// TIA Portal V18 export
FUNCTION_BLOCK "ST10_Flow6_ToolCodeScan"   // FB1076, GRAPH
// stored: AcknowledgeErrorsRequired false, AutoNumber false, GraphVersion 6.0, InitialValuesAcquisition false, SetENOAutomatically false
   // inherited from GRAPH_BASE
   VAR_INPUT
      iSysInface : "RCS_SysComInterface_V1";
   END_VAR
   VAR_IN_OUT
      ioPM_Inface : "RCS_PMInterface_V1";
      ioStatus : Int;
   END_VAR
   VAR
      sCtrlMode { S7_SetPoint := 'True'} : "SysFlowCtrlGraph";
      sUpdMES_Data : Bool;   // 更新MES数据
      工件放行中 : Bool;
      前站站号 { ExternalAccessible := 'False'; ExternalVisible := 'False'; ExternalWritable := 'False'} : UInt;
      本站站号 { ExternalAccessible := 'False'; ExternalVisible := 'False'; ExternalWritable := 'False'} : UInt;
      弹窗Temp : Array[1..10] of Int;
      AlarmID : Int;
      TON { S7_SetPoint := 'True'} : Array[0..10] of TON_TIME;
      TOF { S7_SetPoint := 'True'} : Array[0..10] of TOF_TIME;
      sUP { S7_SetPoint := 'True'} : Array[0..10] of Bool;
      更新RFID完成 : Bool;
   END_VAR
   VAR_TEMP
      Tempresult : USInt;
      本站站号乘10 : UInt;
   END_VAR
   // // TON[0] : 托盘流入1托盘到位传感器 / iA-Rotating product Check
   // // TON[1] : 托盘流入1托盘到位传感器
   // // TON[2] : 托盘流入1产品有无传感器
   // // TON[3] : 托盘流入1产品有无传感器
   // // TON[4] : 托盘流入1姿态检测光电2
   // // TON[5] : 托盘流入1姿态检测光电3
   // // TON[0].Q : 托盘流入1托盘到位 / iA-Rotating product Check
   // // TON[1].Q : 托盘流入1托盘无
   // // TON[2].Q : 托盘流入1有产品
   // // TON[3].Q : 托盘流入1无产品
   // // TON[4].Q : 托盘流入1姿态检测光电2
   // // TON[5].Q : 托盘流入1姿态检测光电3
   // // TOF[1] : iA-Rotating product Check
BEGIN
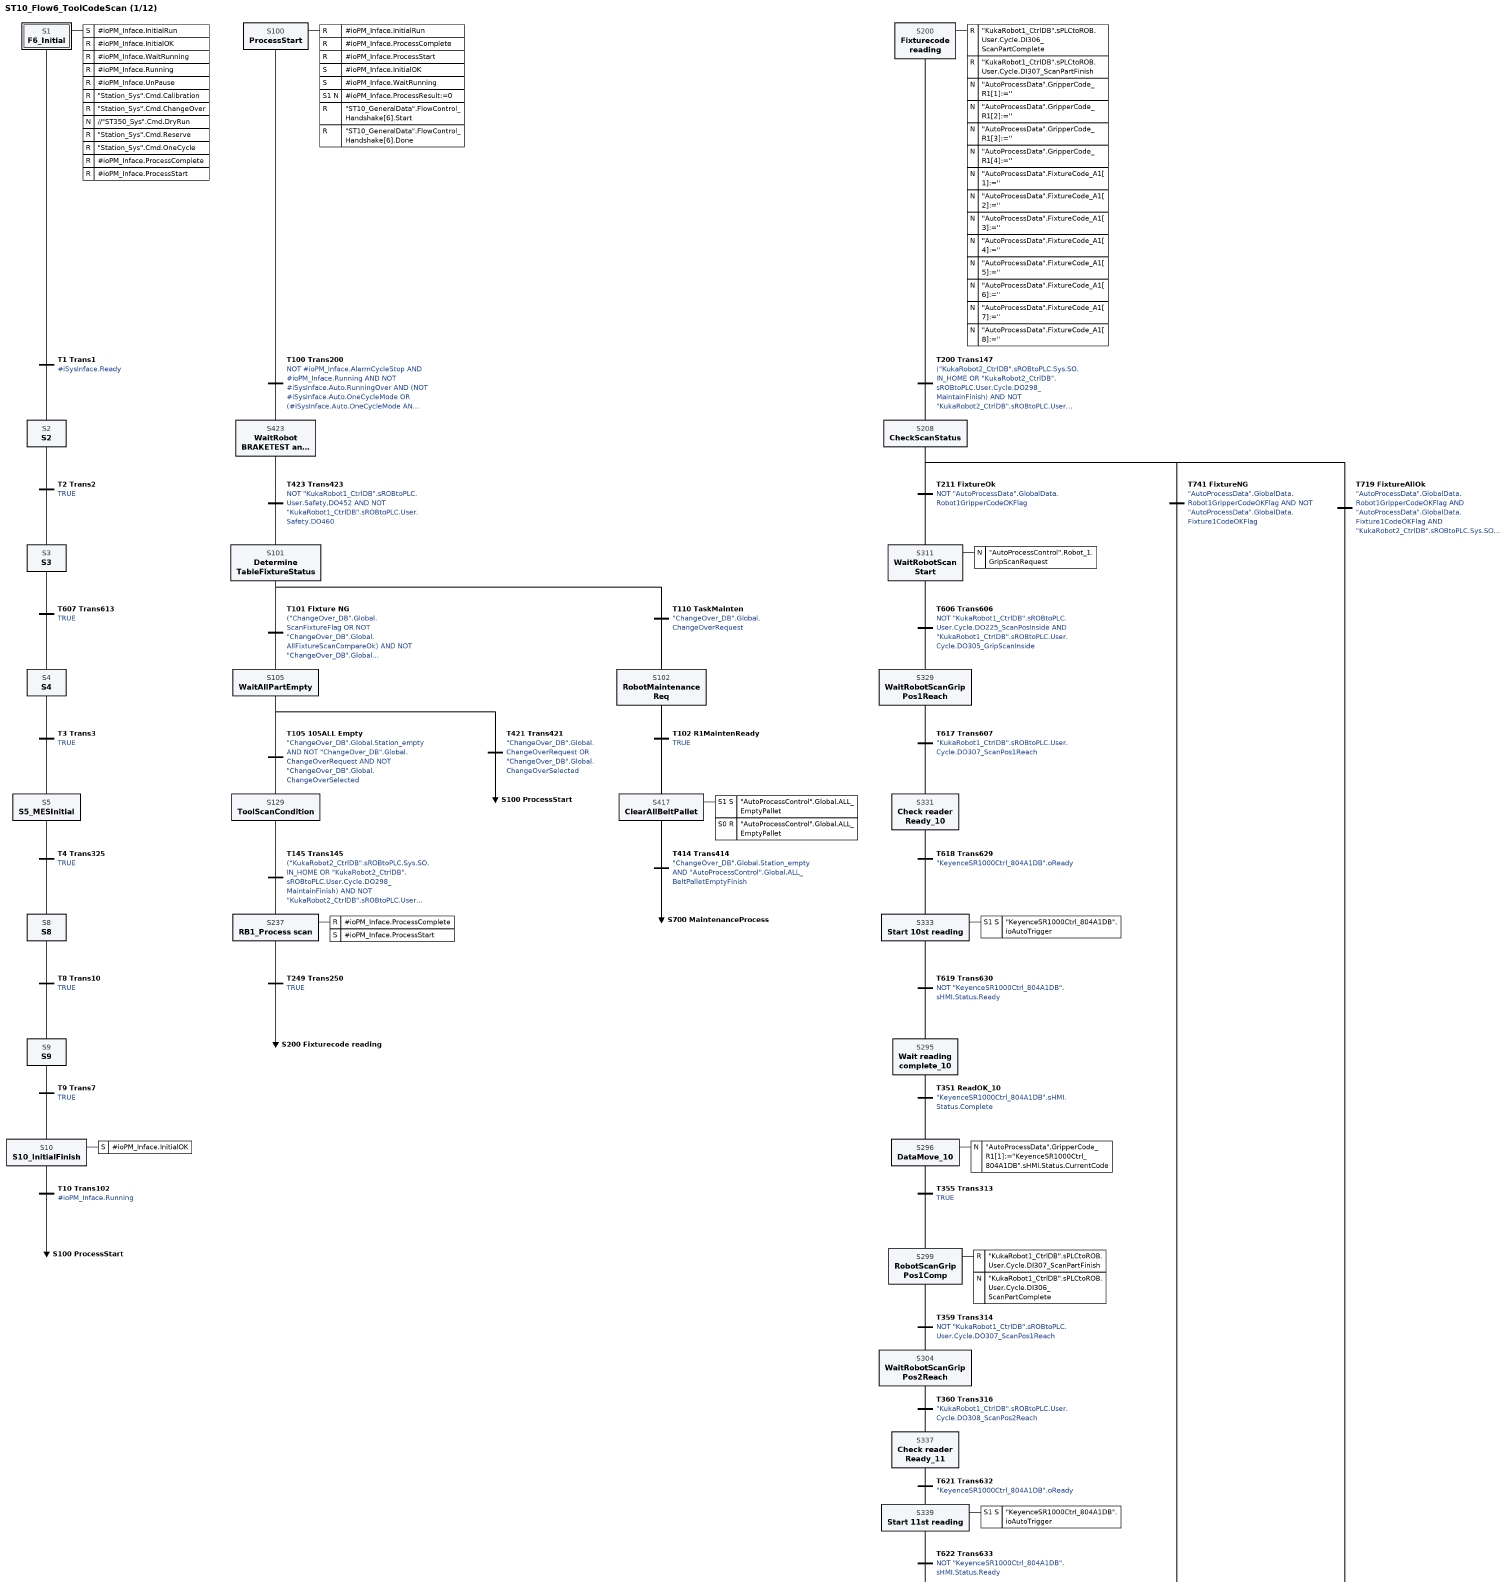
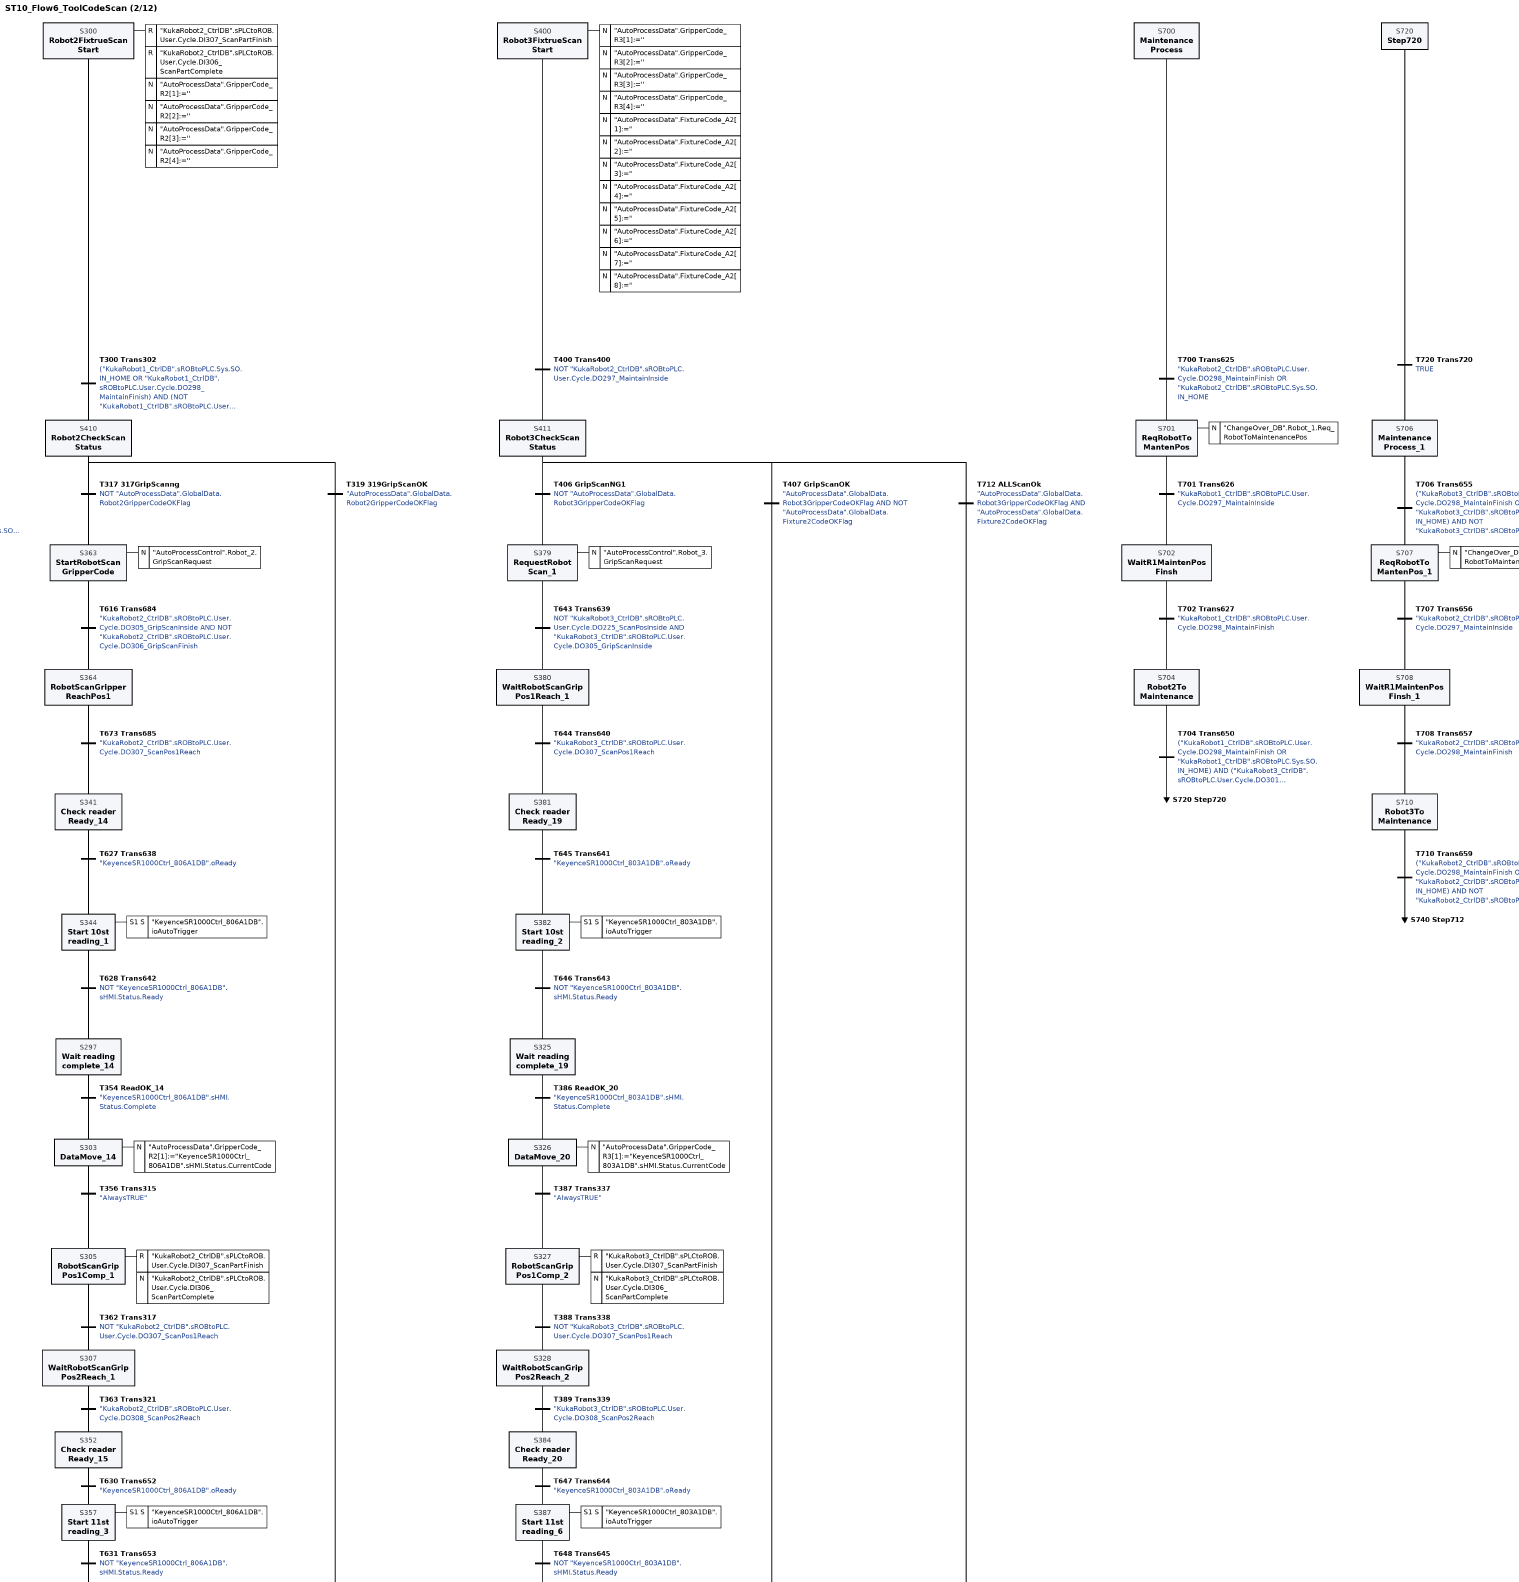
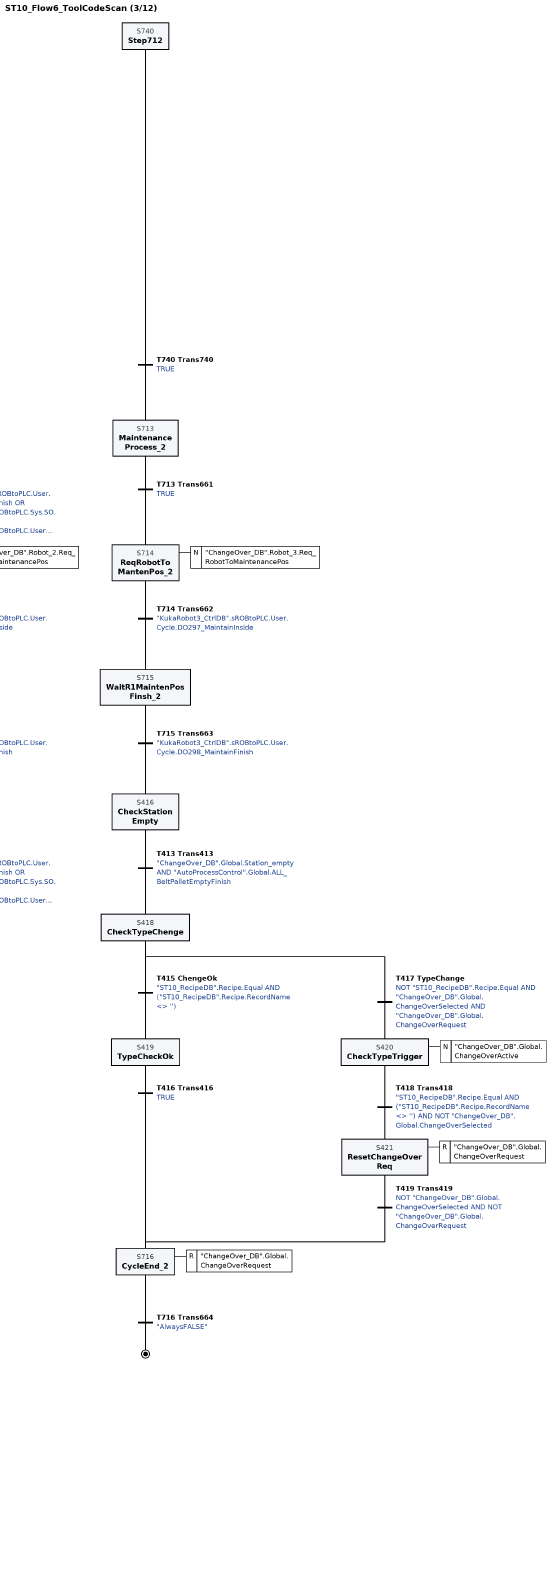
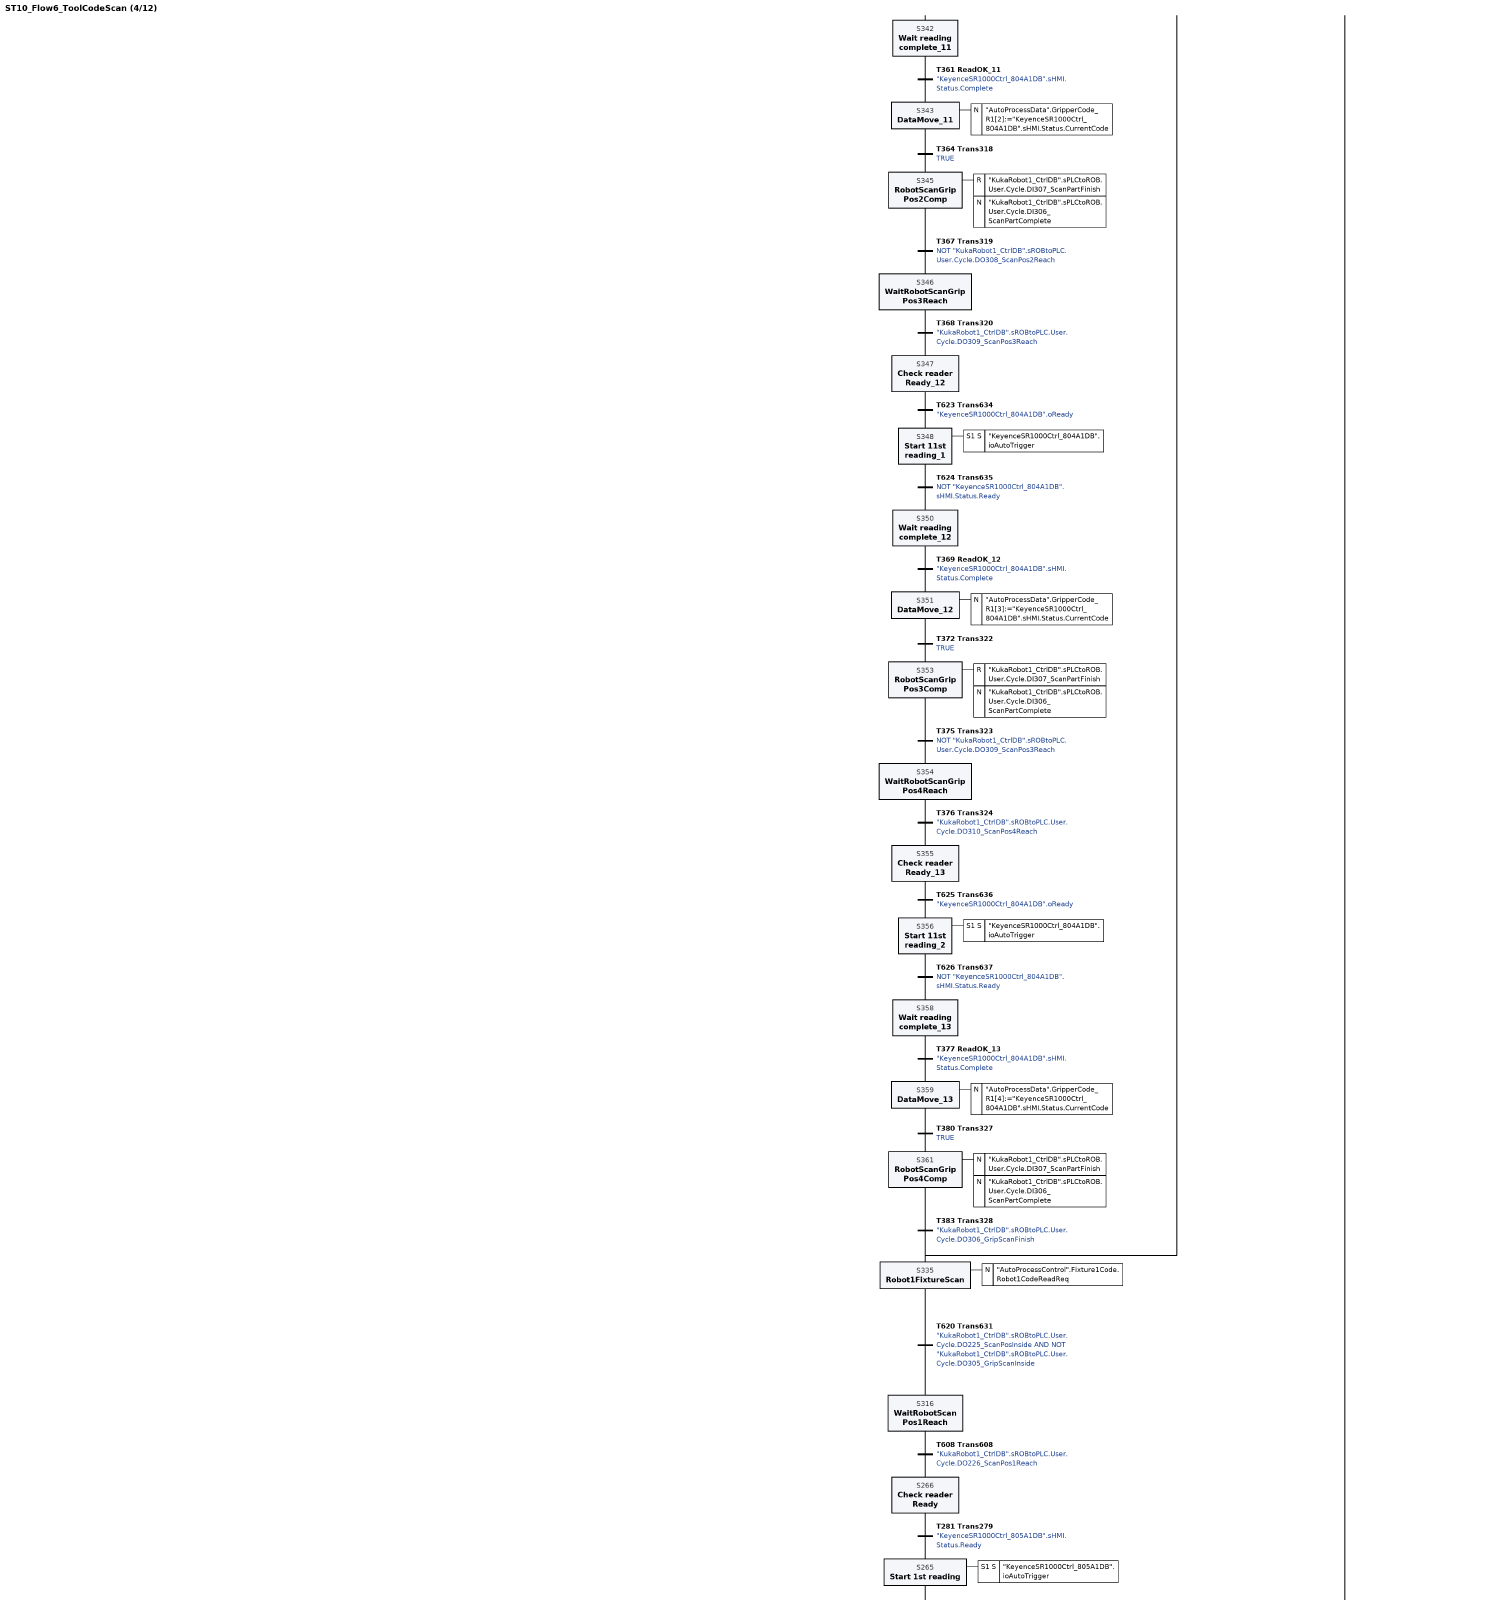
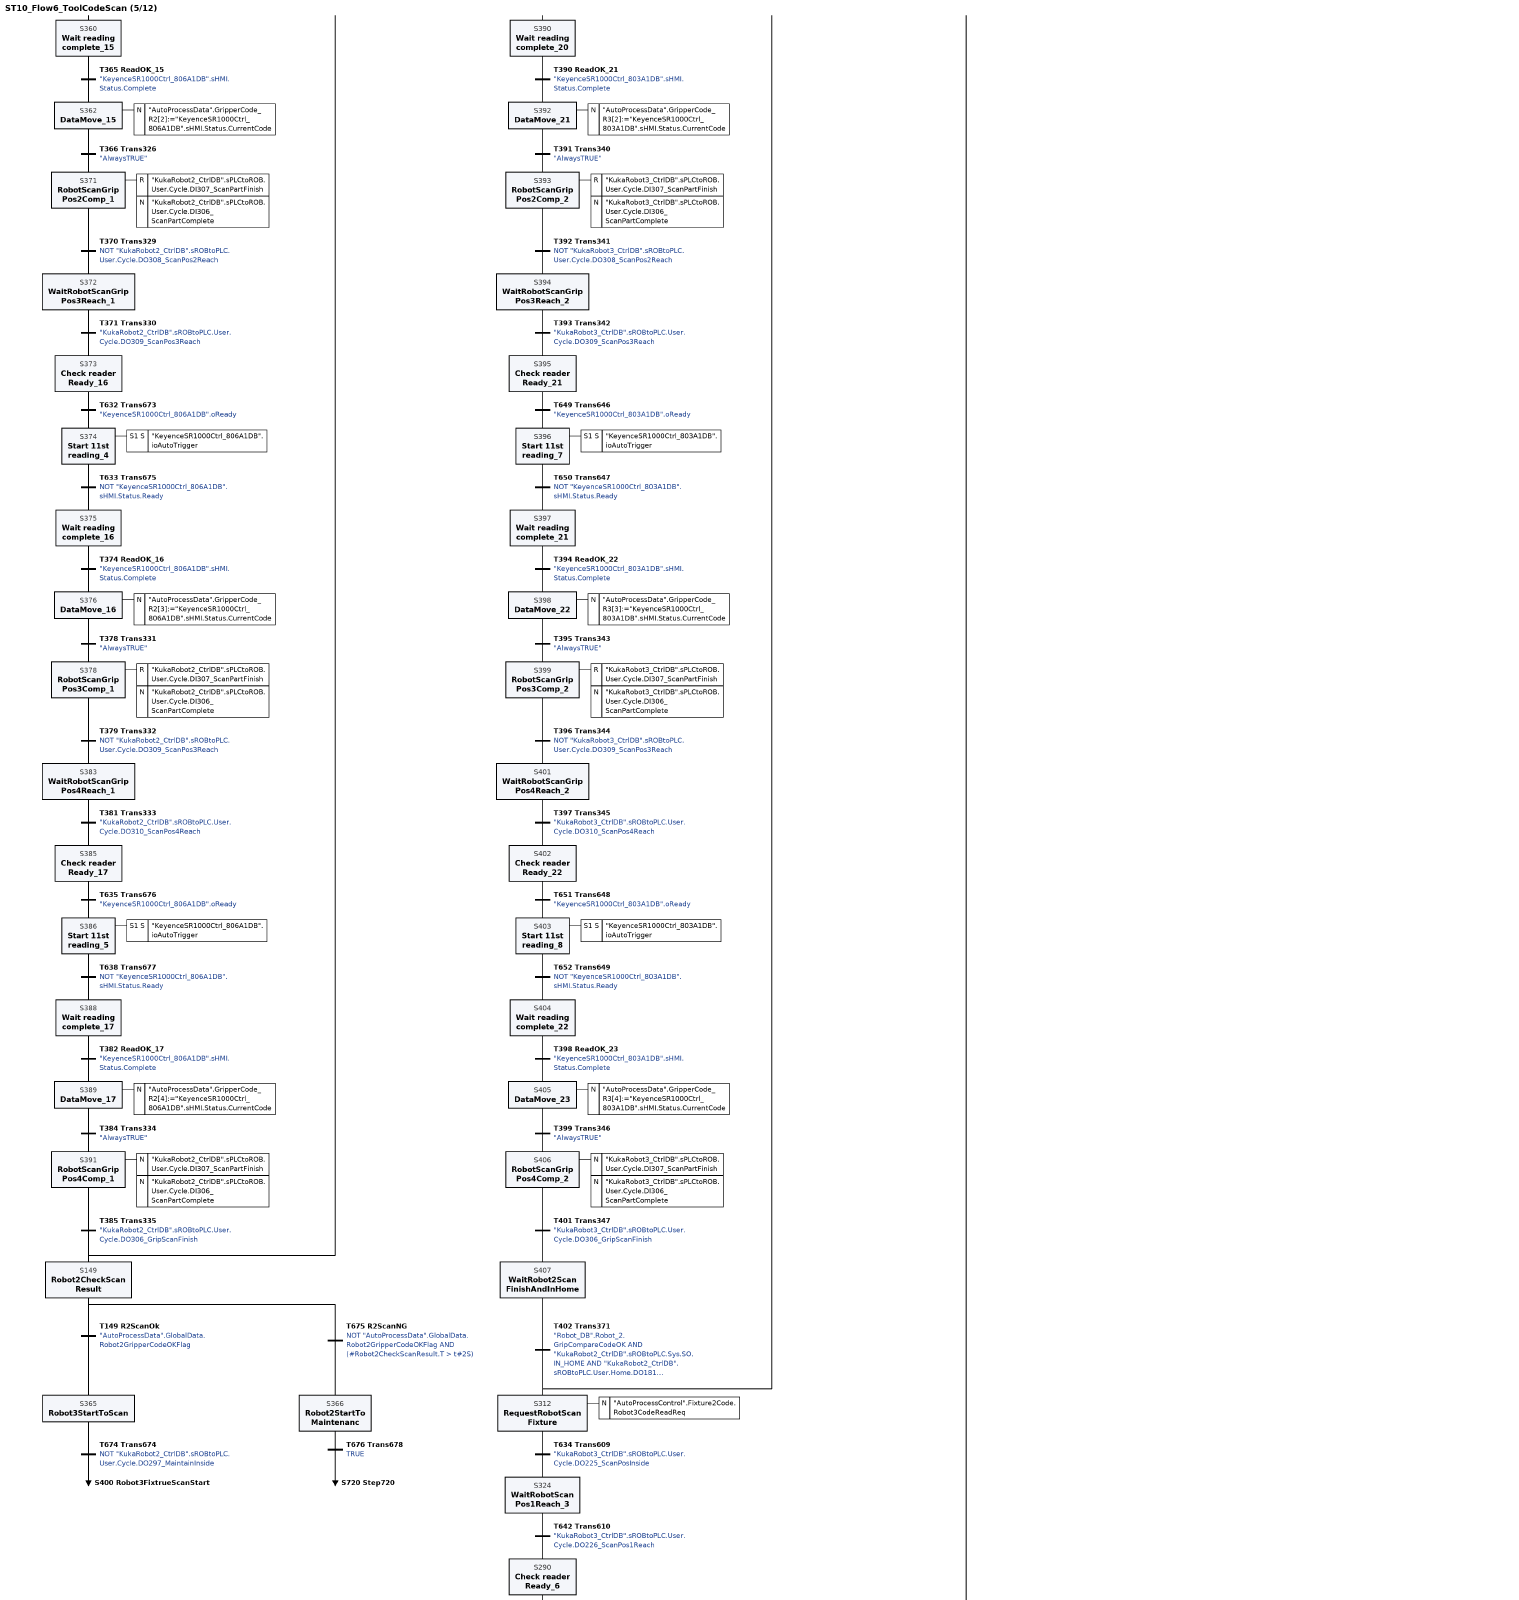
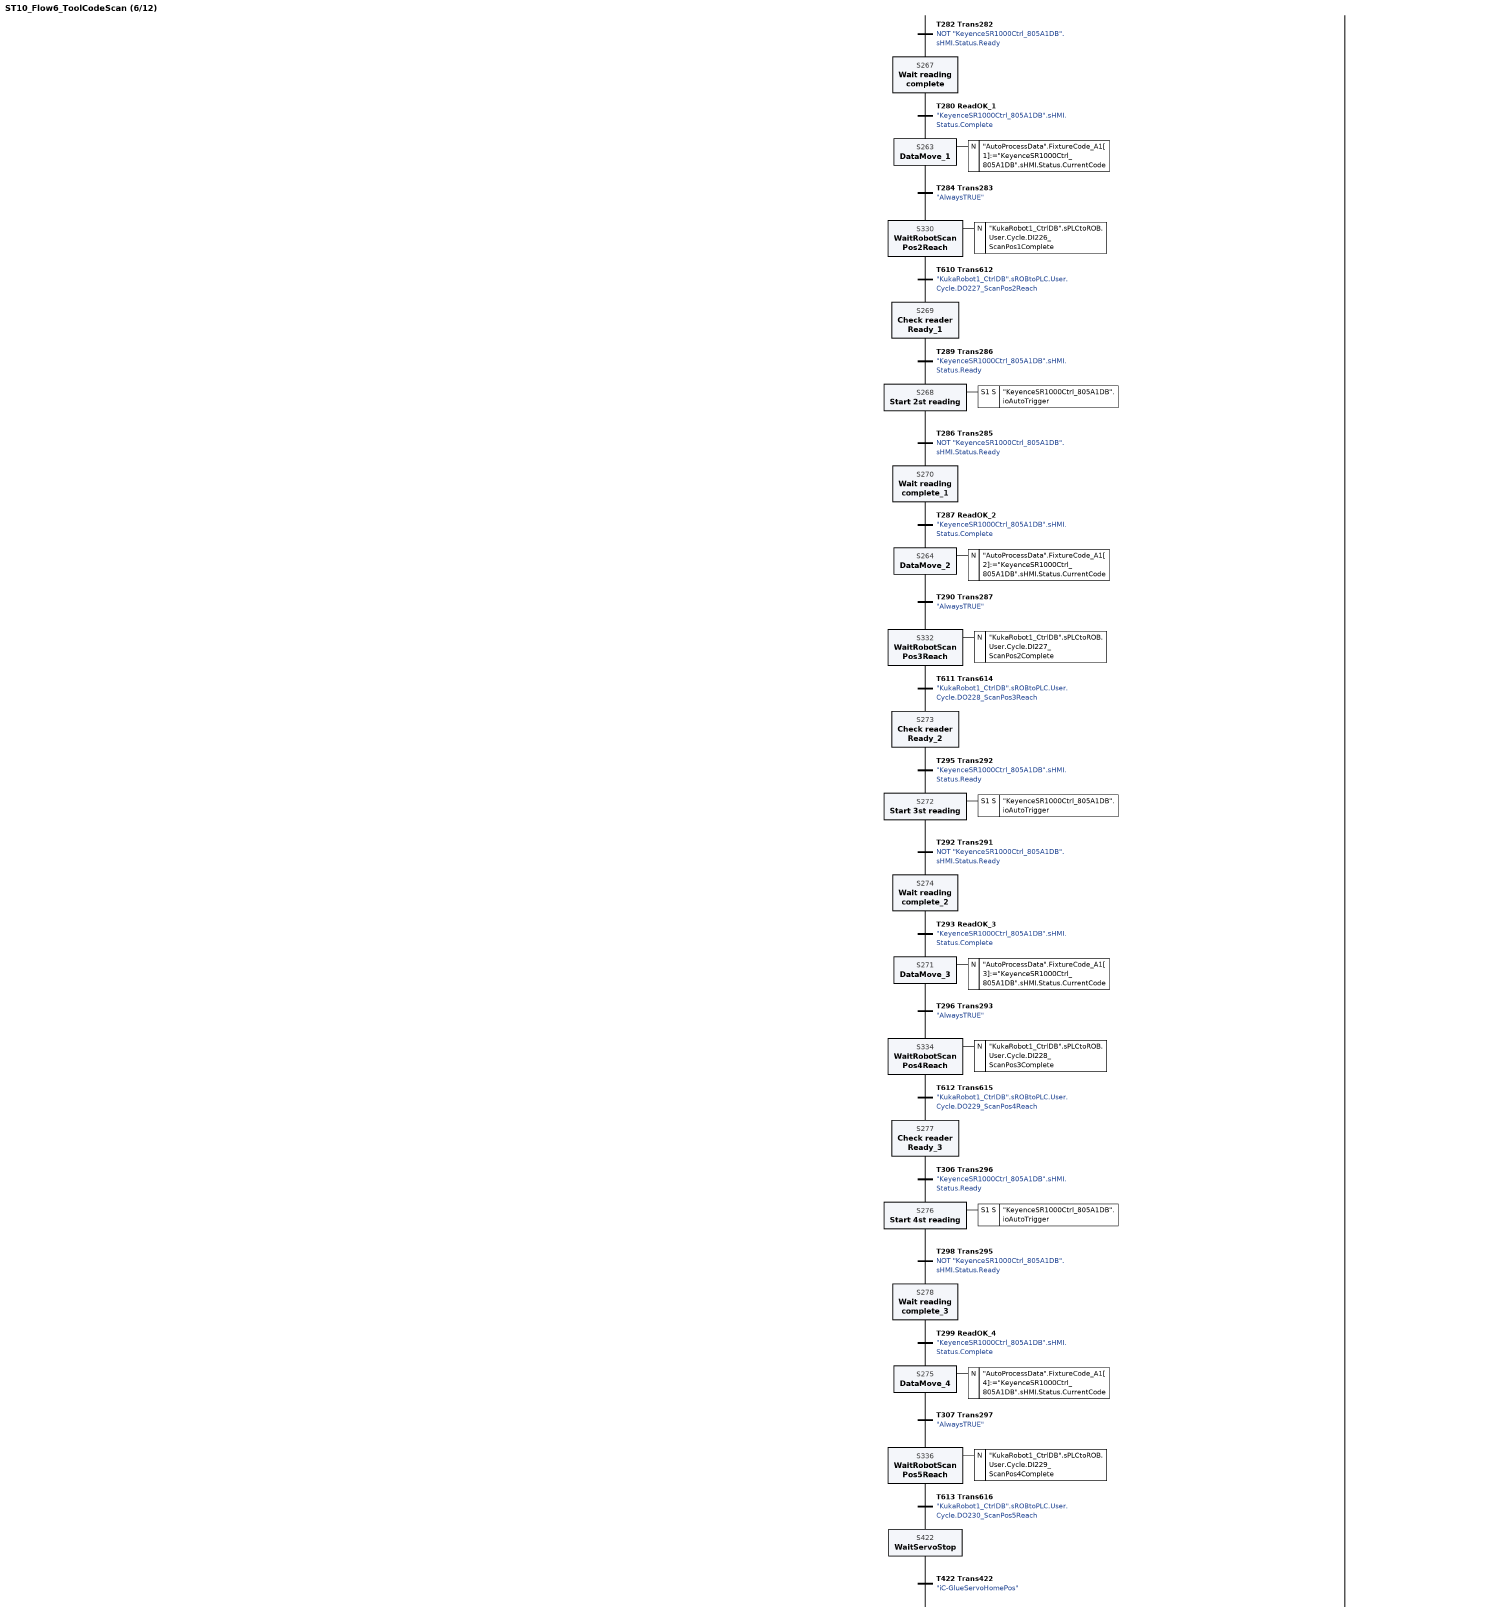
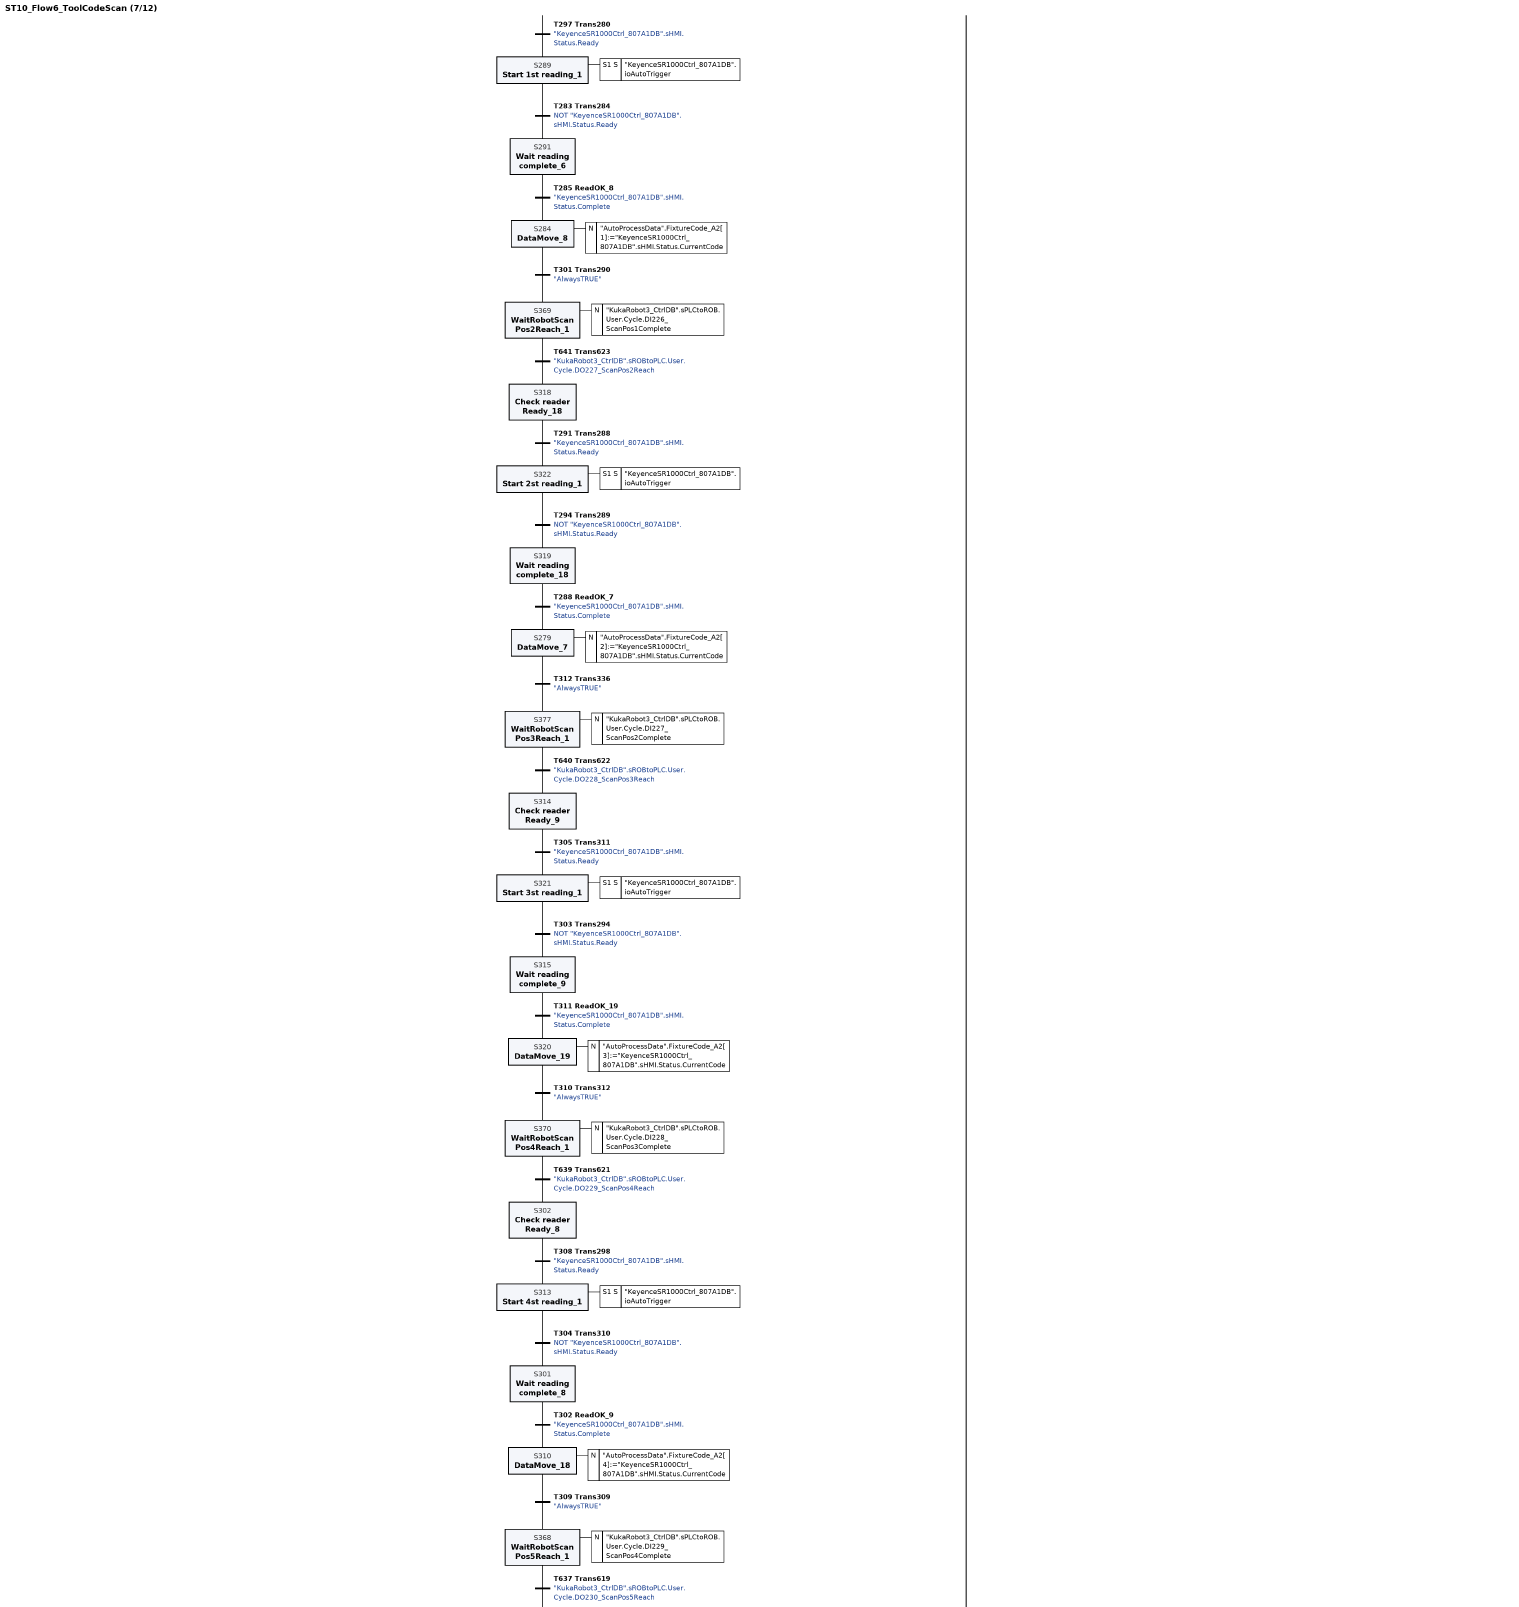
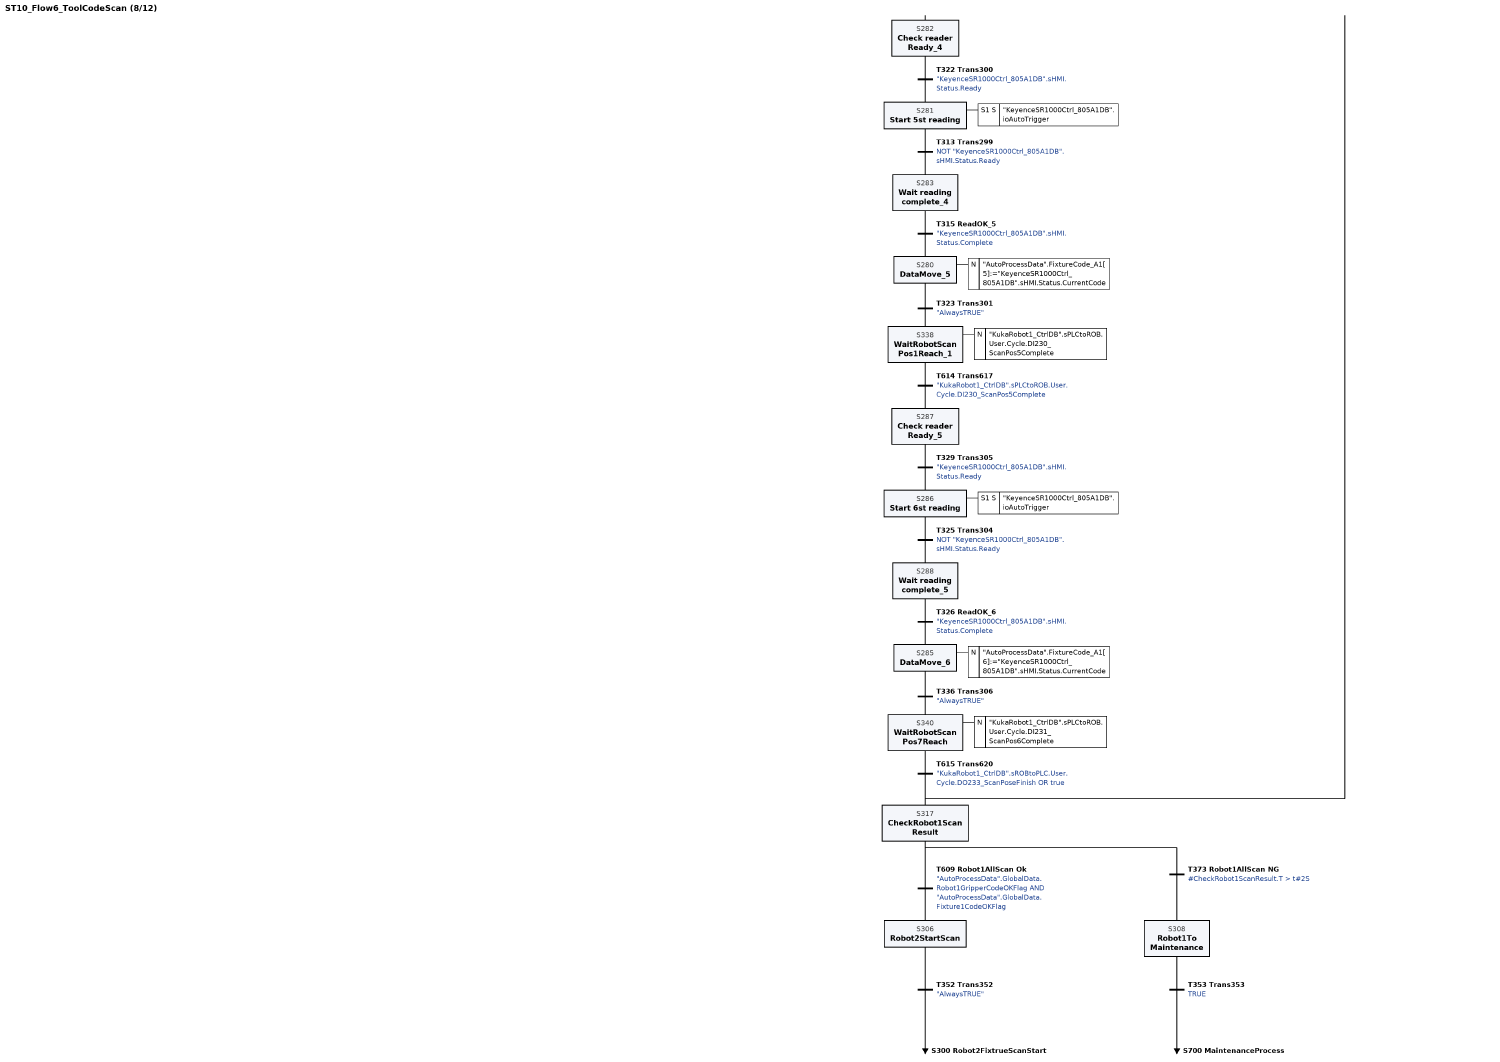
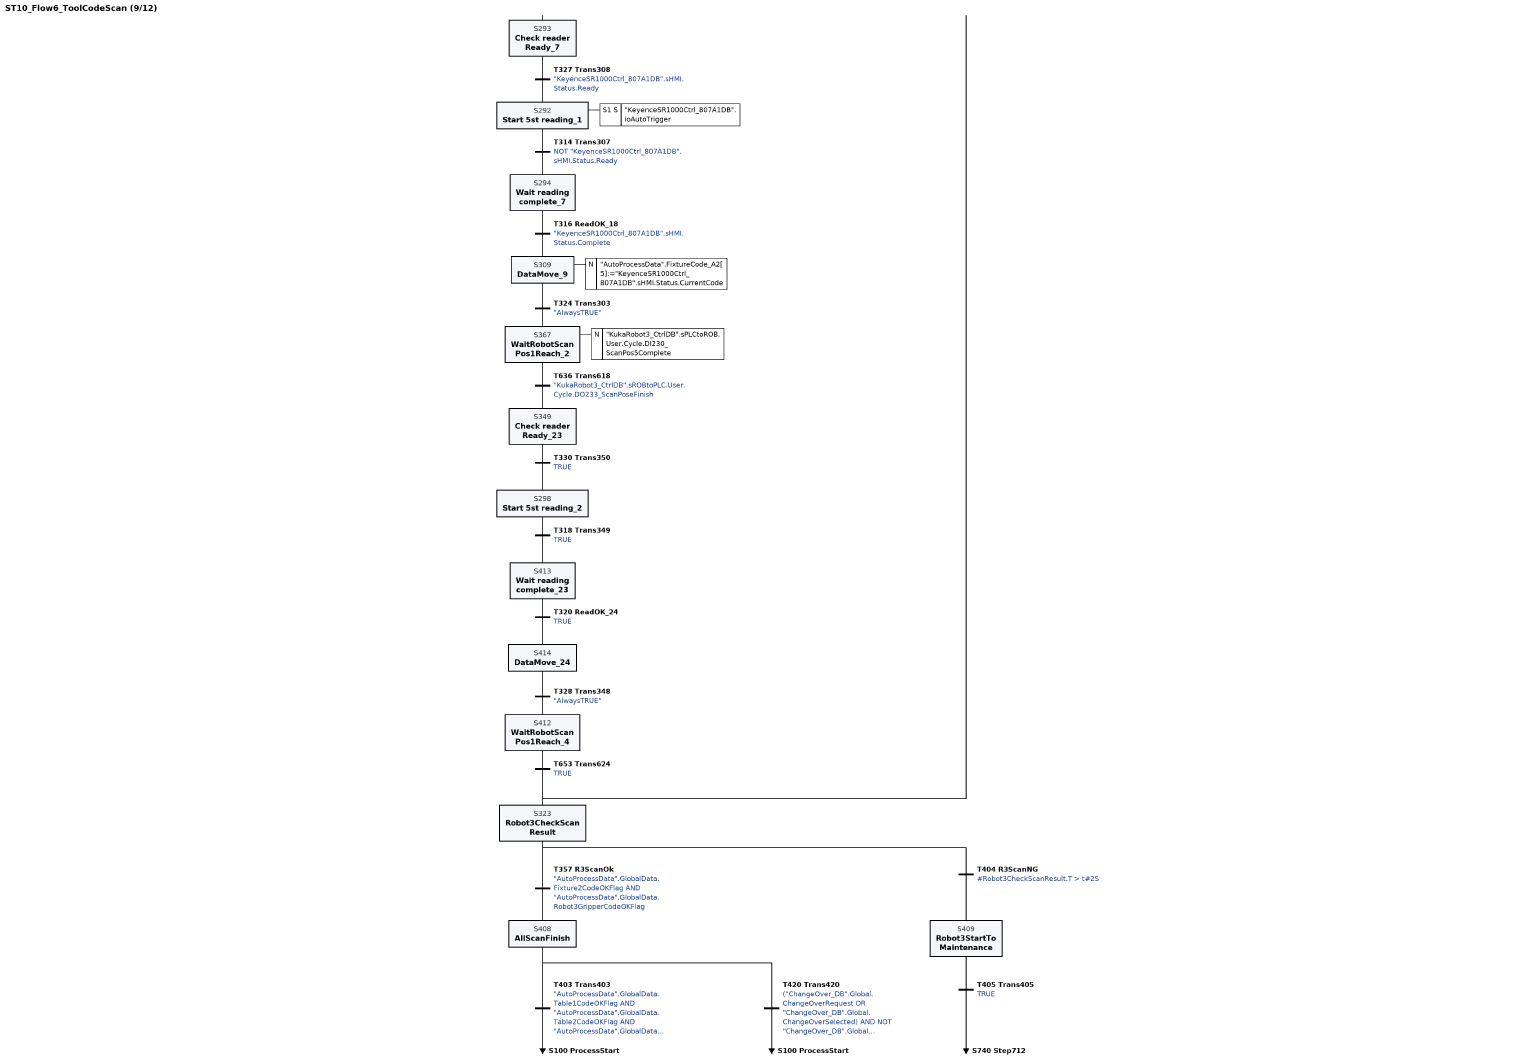
   // permanent pre-instructions
   NETWORK 1
      #TON[10].TON(IN := "AlwaysTRUE" AND "Station_Sys".Alarm.ImmediatelyStop, PT := T#300ms);
      #ioPM_Inface.AlarmImdilyStop := #TON[10].Q;
      #ioPM_Inface.AlarmCycleStop := "AlwaysTRUE" AND "Station_Sys".Alarm.CycleStop;
   NETWORK 2
      IF NOT False THEN
          #sCtrlMode(iSysInface := #iSysInface, ioPM_Inface := #ioPM_Inface, ioGraphCtrl := #RT_DATA.MOP);   // "SysFlowCtrlGraph"
      END_IF;
   NETWORK 3
      #TON[0].TON(IN := "AlwaysTRUE" AND "iA-Rotating product Check", PT := t#500ms);   // 工位11有托盘
      #TON[1].TOF(IN := "AlwaysTRUE" AND NOT "iA-Rotating product Check", PT := T#300ms);   // 工位无托盘
      #TON[2].TON(IN := "AlwaysTRUE", PT := T#300ms);
      #TON[3].TON(IN := "AlwaysTRUE", PT := T#300ms);
      #TON[4].TON(IN := "AlwaysTRUE", PT := T#300ms);
      #TON[5].TON(IN := "AlwaysTRUE", PT := T#300ms);
   NETWORK 4
      #前站站号 := 345;
      #本站站号 := 350;

   // sequencer 1: S01-S99 初始化 / S01-S99 Initial
   INITIAL_STEP F6_Initial:   // S1, max time T#10S, warning time T#7S
              S    #ioPM_Inface.InitialRun
              R    #ioPM_Inface.InitialOK
              R    #ioPM_Inface.WaitRunning
              R    #ioPM_Inface.Running
              R    #ioPM_Inface.UnPause
              R    "Station_Sys".Cmd.Calibration
              R    "Station_Sys".Cmd.ChangeOver
                   //"ST350_Sys".Cmd.DryRun
              R    "Station_Sys".Cmd.Reserve
              R    "Station_Sys".Cmd.OneCycle
              R    #ioPM_Inface.ProcessComplete
              R    #ioPM_Inface.ProcessStart
   END_STEP
   TRANSITION Trans1 FROM F6_Initial TO S2   // T1
      := #iSysInface.Ready;
   END_TRANSITION
   STEP S2:   // S2, max time T#10S, warning time T#7S
   END_STEP
   TRANSITION Trans2 FROM S2 TO S3   // T2
      := TRUE;
   END_TRANSITION
   STEP S4:   // S4, max time T#10S, warning time T#7S
   END_STEP
   TRANSITION Trans3 FROM S4 TO S5_MESInitial   // T3
      := TRUE;
   END_TRANSITION
   STEP S5_MESInitial:   // S5, max time T#10S, warning time T#7S
   END_STEP
   TRANSITION Trans325 FROM S5_MESInitial TO S8   // T4
      := TRUE;
   END_TRANSITION
   STEP S10_InitialFinish:   // S10, max time T#10S, warning time T#7S
              S    #ioPM_Inface.InitialOK
   END_STEP
   TRANSITION Trans102 FROM S10_InitialFinish TO ProcessStart   // T10, jump
      := #ioPM_Inface.Running;
   END_TRANSITION
   STEP S3:   // S3, max time T#10S, warning time T#7S
   END_STEP
   TRANSITION Trans613 FROM S3 TO S4   // T607
      := TRUE;
   END_TRANSITION
   STEP S8:   // S8, max time T#10S, warning time T#7S
   END_STEP
   TRANSITION Trans10 FROM S8 TO S9   // T8
      := TRUE;
   END_TRANSITION
   STEP S9:   // S9, max time T#10S, warning time T#7S
   END_STEP
   TRANSITION Trans7 FROM S9 TO S10_InitialFinish   // T9
      := TRUE;
   END_TRANSITION

   // sequencer 2: S100-S199 等待到位 / S100-S199 Fixture Scan Task
   STEP ProcessStart:   // S100, max time T#10S, warning time T#7S
      // 自动等待开始运行
              R    #ioPM_Inface.InitialRun
              R    #ioPM_Inface.ProcessComplete
              R    #ioPM_Inface.ProcessStart
              S    #ioPM_Inface.InitialOK
              S    #ioPM_Inface.WaitRunning
          S1  N    #ioPM_Inface.ProcessResult:=0
              R    "ST10_GeneralData".FlowControl_Handshake[6].Start
              R    "ST10_GeneralData".FlowControl_Handshake[6].Done
   END_STEP
   TRANSITION Trans200 FROM ProcessStart TO "WaitRobotBRAKETEST and MASTERINGTEST finish"   // T100
      := NOT #ioPM_Inface.AlarmCycleStop AND #ioPM_Inface.Running AND NOT #iSysInface.Auto.RunningOver AND (NOT #iSysInface.Auto.OneCycleMode OR (#iSysInface.Auto.OneCycleMode AND #ioPM_Inface.TriggerOneCycle));
   END_TRANSITION
   STEP "RB1_Process scan":   // S237, max time T#10S, warning time T#7S
              R    #ioPM_Inface.ProcessComplete
              S    #ioPM_Inface.ProcessStart
   END_STEP
   TRANSITION Trans250 FROM "RB1_Process scan" TO "Fixturecode reading"   // T249, jump
      := TRUE;
   END_TRANSITION
   STEP "Determine TableFixtureStatus":   // S101, max time T#10S, warning time T#7S
   END_STEP
   TRANSITION "Fixture NG" FROM "Determine TableFixtureStatus" TO WaitAllPartEmpty   // T101
      := ("ChangeOver_DB".Global.ScanFixtureFlag OR NOT "ChangeOver_DB".Global.AllFixtureScanCompareOk) AND NOT "ChangeOver_DB".Global.ChangeOverRequest AND NOT "ChangeOver_DB".Global.ChangeOverSelected;
   END_TRANSITION
   TRANSITION TaskMainten FROM "Determine TableFixtureStatus" TO RobotMaintenanceReq   // T110
      := "ChangeOver_DB".Global.ChangeOverRequest;
   END_TRANSITION
   STEP RobotMaintenanceReq:   // S102, max time T#10S, warning time T#7S
   END_STEP
   TRANSITION R1MaintenReady FROM RobotMaintenanceReq TO ClearAllBeltPallet   // T102
      := TRUE;
   END_TRANSITION
   STEP ToolScanCondition:   // S129, max time T#10S, warning time T#7S
   END_STEP
   TRANSITION Trans145 FROM ToolScanCondition TO "RB1_Process scan"   // T145
      := ("KukaRobot2_CtrlDB".sROBtoPLC.Sys.SO.IN_HOME OR "KukaRobot2_CtrlDB".sROBtoPLC.User.Cycle.DO298_MaintainFinish) AND NOT "KukaRobot2_CtrlDB".sROBtoPLC.User.Cycle.DO305_GripScanInside;
   END_TRANSITION
   STEP ClearAllBeltPallet:   // S417, max time T#10S, warning time T#7S
          S1  S    "AutoProcessControl".Global.ALL_EmptyPallet
          S0  R    "AutoProcessControl".Global.ALL_EmptyPallet
   END_STEP
   TRANSITION Trans414 FROM ClearAllBeltPallet TO MaintenanceProcess   // T414, jump
      := "ChangeOver_DB".Global.Station_empty AND "AutoProcessControl".Global.ALL_BeltPalletEmptyFinish;
   END_TRANSITION
   STEP WaitAllPartEmpty:   // S105, max time T#10S, warning time T#7S
   END_STEP
   TRANSITION "105ALL Empty" FROM WaitAllPartEmpty TO ToolScanCondition   // T105
      := "ChangeOver_DB".Global.Station_empty AND NOT "ChangeOver_DB".Global.ChangeOverRequest AND NOT "ChangeOver_DB".Global.ChangeOverSelected;
   END_TRANSITION
   TRANSITION Trans421 FROM WaitAllPartEmpty TO ProcessStart   // T421, jump
      := "ChangeOver_DB".Global.ChangeOverRequest OR "ChangeOver_DB".Global.ChangeOverSelected;
   END_TRANSITION
   STEP "WaitRobotBRAKETEST and MASTERINGTEST finish":   // S423, max time T#10S, warning time T#7S
   END_STEP
   TRANSITION Trans423 FROM "WaitRobotBRAKETEST and MASTERINGTEST finish" TO "Determine TableFixtureStatus"   // T423
      := NOT "KukaRobot1_CtrlDB".sROBtoPLC.User.Safety.DO452 AND NOT "KukaRobot1_CtrlDB".sROBtoPLC.User.Safety.DO460;
   END_TRANSITION

   // sequencer 3: S200-S299 Robot1 FixtureCode reading
   STEP "Fixturecode reading":   // S200, max time T#10S, warning time T#7S
              R    "KukaRobot1_CtrlDB".sPLCtoROB.User.Cycle.DI306_ScanPartComplete
              R    "KukaRobot1_CtrlDB".sPLCtoROB.User.Cycle.DI307_ScanPartFinish
              N    "AutoProcessData".GripperCode_R1[1]:=''
              N    "AutoProcessData".GripperCode_R1[2]:=''
              N    "AutoProcessData".GripperCode_R1[3]:=''
              N    "AutoProcessData".GripperCode_R1[4]:=''
              N    "AutoProcessData".FixtureCode_A1[1]:=''
              N    "AutoProcessData".FixtureCode_A1[2]:=''
              N    "AutoProcessData".FixtureCode_A1[3]:=''
              N    "AutoProcessData".FixtureCode_A1[4]:=''
              N    "AutoProcessData".FixtureCode_A1[5]:=''
              N    "AutoProcessData".FixtureCode_A1[6]:=''
              N    "AutoProcessData".FixtureCode_A1[7]:=''
              N    "AutoProcessData".FixtureCode_A1[8]:=''
   END_STEP
   TRANSITION Trans147 FROM "Fixturecode reading" TO CheckScanStatus   // T200
      := ("KukaRobot2_CtrlDB".sROBtoPLC.Sys.SO.IN_HOME OR "KukaRobot2_CtrlDB".sROBtoPLC.User.Cycle.DO298_MaintainFinish) AND NOT "KukaRobot2_CtrlDB".sROBtoPLC.User.Cycle.DO305_GripScanInside;
   END_TRANSITION
   STEP DataMove_2:   // S264, max time T#10S, warning time T#7S
              N    "AutoProcessData".FixtureCode_A1[2]:="KeyenceSR1000Ctrl_805A1DB".sHMI.Status.CurrentCode
   END_STEP
   TRANSITION Trans287 FROM DataMove_2 TO WaitRobotScanPos3Reach   // T290
      := "AlwaysTRUE";
   END_TRANSITION
   STEP Robot1ToMaintenance:   // S308, max time T#10S, warning time T#7S
   END_STEP
   TRANSITION Trans353 FROM Robot1ToMaintenance TO MaintenanceProcess   // T353, jump
      := TRUE;
   END_TRANSITION
   STEP CheckScanStatus:   // S208, max time T#10S, warning time T#7S
   END_STEP
   TRANSITION FixtureOk FROM CheckScanStatus TO WaitRobotScanStart   // T211
      := NOT "AutoProcessData".GlobalData.Robot1GripperCodeOKFlag;
   END_TRANSITION
   TRANSITION FixtureNG FROM CheckScanStatus TO Robot1FixtureScan   // T741
      := "AutoProcessData".GlobalData.Robot1GripperCodeOKFlag AND NOT "AutoProcessData".GlobalData.Fixture1CodeOKFlag;
   END_TRANSITION
   TRANSITION FixtureAllOk FROM CheckScanStatus TO CheckRobot1ScanResult   // T719
      := "AutoProcessData".GlobalData.Robot1GripperCodeOKFlag AND "AutoProcessData".GlobalData.Fixture1CodeOKFlag AND "KukaRobot2_CtrlDB".sROBtoPLC.Sys.SO.IN_HOME AND NOT "KukaRobot2_CtrlDB".sROBtoPLC.User.Cycle.DO305_GripScanInside;
   END_TRANSITION
   STEP DataMove_1:   // S263, max time T#10S, warning time T#7S
              N    "AutoProcessData".FixtureCode_A1[1]:="KeyenceSR1000Ctrl_805A1DB".sHMI.Status.CurrentCode
   END_STEP
   TRANSITION Trans283 FROM DataMove_1 TO WaitRobotScanPos2Reach   // T284
      := "AlwaysTRUE";
   END_TRANSITION
   STEP WaitRobotScanStart:   // S311, max time T#10S, warning time T#7S
              N    "AutoProcessControl".Robot_1.GripScanRequest
   END_STEP
   TRANSITION Trans606 FROM WaitRobotScanStart TO WaitRobotScanGripPos1Reach   // T606
      := NOT "KukaRobot1_CtrlDB".sROBtoPLC.User.Cycle.DO225_ScanPosInside AND "KukaRobot1_CtrlDB".sROBtoPLC.User.Cycle.DO305_GripScanInside;
   END_TRANSITION
   STEP "Start 1st reading":   // S265, max time T#10S, warning time T#7S
          S1  S    "KeyenceSR1000Ctrl_805A1DB".ioAutoTrigger
   END_STEP
   TRANSITION Trans282 FROM "Start 1st reading" TO "Wait reading complete"   // T282
      := NOT "KeyenceSR1000Ctrl_805A1DB".sHMI.Status.Ready;
   END_TRANSITION
   STEP "Check reader Ready":   // S266, max time T#10S, warning time T#7S
   END_STEP
   TRANSITION Trans279 FROM "Check reader Ready" TO "Start 1st reading"   // T281
      := "KeyenceSR1000Ctrl_805A1DB".sHMI.Status.Ready;
   END_TRANSITION
   STEP "Wait reading complete":   // S267, max time T#10S, warning time T#7S
   END_STEP
   TRANSITION ReadOK_1 FROM "Wait reading complete" TO DataMove_1   // T280
      := "KeyenceSR1000Ctrl_805A1DB".sHMI.Status.Complete;
   END_TRANSITION
   STEP "Wait reading complete_5":   // S288, max time T#10S, warning time T#7S
   END_STEP
   TRANSITION ReadOK_6 FROM "Wait reading complete_5" TO DataMove_6   // T326
      := "KeyenceSR1000Ctrl_805A1DB".sHMI.Status.Complete;
   END_TRANSITION
   STEP "Check reader Ready_5":   // S287, max time T#10S, warning time T#7S
   END_STEP
   TRANSITION Trans305 FROM "Check reader Ready_5" TO "Start 6st reading"   // T329
      := "KeyenceSR1000Ctrl_805A1DB".sHMI.Status.Ready;
   END_TRANSITION
   STEP "Start 6st reading":   // S286, max time T#10S, warning time T#7S
          S1  S    "KeyenceSR1000Ctrl_805A1DB".ioAutoTrigger
   END_STEP
   TRANSITION Trans304 FROM "Start 6st reading" TO "Wait reading complete_5"   // T325
      := NOT "KeyenceSR1000Ctrl_805A1DB".sHMI.Status.Ready;
   END_TRANSITION
   STEP WaitRobotScanPos1Reach_1:   // S338, max time T#10S, warning time T#7S
              N    "KukaRobot1_CtrlDB".sPLCtoROB.User.Cycle.DI230_ScanPos5Complete
   END_STEP
   TRANSITION Trans617 FROM WaitRobotScanPos1Reach_1 TO "Check reader Ready_5"   // T614
      := "KukaRobot1_CtrlDB".sPLCtoROB.User.Cycle.DI230_ScanPos5Complete;
   END_TRANSITION
   STEP WaitRobotScanPos5Reach:   // S336, max time T#10S, warning time T#7S
              N    "KukaRobot1_CtrlDB".sPLCtoROB.User.Cycle.DI229_ScanPos4Complete
   END_STEP
   TRANSITION Trans616 FROM WaitRobotScanPos5Reach TO WaitServoStop   // T613
      := "KukaRobot1_CtrlDB".sROBtoPLC.User.Cycle.DO230_ScanPos5Reach;
   END_TRANSITION
   STEP DataMove_6:   // S285, max time T#10S, warning time T#7S
              N    "AutoProcessData".FixtureCode_A1[6]:="KeyenceSR1000Ctrl_805A1DB".sHMI.Status.CurrentCode
   END_STEP
   TRANSITION Trans306 FROM DataMove_6 TO WaitRobotScanPos7Reach   // T336
      := "AlwaysTRUE";
   END_TRANSITION
   STEP WaitRobotScanPos2Reach:   // S330, max time T#10S, warning time T#7S
              N    "KukaRobot1_CtrlDB".sPLCtoROB.User.Cycle.DI226_ScanPos1Complete
   END_STEP
   TRANSITION Trans612 FROM WaitRobotScanPos2Reach TO "Check reader Ready_1"   // T610
      := "KukaRobot1_CtrlDB".sROBtoPLC.User.Cycle.DO227_ScanPos2Reach;
   END_TRANSITION
   STEP WaitRobotScanPos4Reach:   // S334, max time T#10S, warning time T#7S
              N    "KukaRobot1_CtrlDB".sPLCtoROB.User.Cycle.DI228_ScanPos3Complete
   END_STEP
   TRANSITION Trans615 FROM WaitRobotScanPos4Reach TO "Check reader Ready_3"   // T612
      := "KukaRobot1_CtrlDB".sROBtoPLC.User.Cycle.DO229_ScanPos4Reach;
   END_TRANSITION
   STEP "Start 5st reading":   // S281, max time T#10S, warning time T#7S
          S1  S    "KeyenceSR1000Ctrl_805A1DB".ioAutoTrigger
   END_STEP
   TRANSITION Trans299 FROM "Start 5st reading" TO "Wait reading complete_4"   // T313
      := NOT "KeyenceSR1000Ctrl_805A1DB".sHMI.Status.Ready;
   END_TRANSITION
   STEP "Check reader Ready_4":   // S282, max time T#10S, warning time T#7S
   END_STEP
   TRANSITION Trans300 FROM "Check reader Ready_4" TO "Start 5st reading"   // T322
      := "KeyenceSR1000Ctrl_805A1DB".sHMI.Status.Ready;
   END_TRANSITION
   STEP "Wait reading complete_4":   // S283, max time T#10S, warning time T#7S
   END_STEP
   TRANSITION ReadOK_5 FROM "Wait reading complete_4" TO DataMove_5   // T315
      := "KeyenceSR1000Ctrl_805A1DB".sHMI.Status.Complete;
   END_TRANSITION
   STEP "Wait reading complete_3":   // S278, max time T#10S, warning time T#7S
   END_STEP
   TRANSITION ReadOK_4 FROM "Wait reading complete_3" TO DataMove_4   // T299
      := "KeyenceSR1000Ctrl_805A1DB".sHMI.Status.Complete;
   END_TRANSITION
   STEP "Check reader Ready_3":   // S277, max time T#10S, warning time T#7S
   END_STEP
   TRANSITION Trans296 FROM "Check reader Ready_3" TO "Start 4st reading"   // T306
      := "KeyenceSR1000Ctrl_805A1DB".sHMI.Status.Ready;
   END_TRANSITION
   STEP DataMove_5:   // S280, max time T#10S, warning time T#7S
              N    "AutoProcessData".FixtureCode_A1[5]:="KeyenceSR1000Ctrl_805A1DB".sHMI.Status.CurrentCode
   END_STEP
   TRANSITION Trans301 FROM DataMove_5 TO WaitRobotScanPos1Reach_1   // T323
      := "AlwaysTRUE";
   END_TRANSITION
   STEP DataMove_4:   // S275, max time T#10S, warning time T#7S
              N    "AutoProcessData".FixtureCode_A1[4]:="KeyenceSR1000Ctrl_805A1DB".sHMI.Status.CurrentCode
   END_STEP
   TRANSITION Trans297 FROM DataMove_4 TO WaitRobotScanPos5Reach   // T307
      := "AlwaysTRUE";
   END_TRANSITION
   STEP "Start 4st reading":   // S276, max time T#10S, warning time T#7S
          S1  S    "KeyenceSR1000Ctrl_805A1DB".ioAutoTrigger
   END_STEP
   TRANSITION Trans295 FROM "Start 4st reading" TO "Wait reading complete_3"   // T298
      := NOT "KeyenceSR1000Ctrl_805A1DB".sHMI.Status.Ready;
   END_TRANSITION
   STEP "Check reader Ready_2":   // S273, max time T#10S, warning time T#7S
   END_STEP
   TRANSITION Trans292 FROM "Check reader Ready_2" TO "Start 3st reading"   // T295
      := "KeyenceSR1000Ctrl_805A1DB".sHMI.Status.Ready;
   END_TRANSITION
   STEP "Wait reading complete_2":   // S274, max time T#10S, warning time T#7S
   END_STEP
   TRANSITION ReadOK_3 FROM "Wait reading complete_2" TO DataMove_3   // T293
      := "KeyenceSR1000Ctrl_805A1DB".sHMI.Status.Complete;
   END_TRANSITION
   STEP WaitRobotScanPos3Reach:   // S332, max time T#10S, warning time T#7S
              N    "KukaRobot1_CtrlDB".sPLCtoROB.User.Cycle.DI227_ScanPos2Complete
   END_STEP
   TRANSITION Trans614 FROM WaitRobotScanPos3Reach TO "Check reader Ready_2"   // T611
      := "KukaRobot1_CtrlDB".sROBtoPLC.User.Cycle.DO228_ScanPos3Reach;
   END_TRANSITION
   STEP "Check reader Ready_1":   // S269, max time T#10S, warning time T#7S
   END_STEP
   TRANSITION Trans286 FROM "Check reader Ready_1" TO "Start 2st reading"   // T289
      := "KeyenceSR1000Ctrl_805A1DB".sHMI.Status.Ready;
   END_TRANSITION
   STEP "Wait reading complete_1":   // S270, max time T#10S, warning time T#7S
   END_STEP
   TRANSITION ReadOK_2 FROM "Wait reading complete_1" TO DataMove_2   // T287
      := "KeyenceSR1000Ctrl_805A1DB".sHMI.Status.Complete;
   END_TRANSITION
   STEP DataMove_3:   // S271, max time T#10S, warning time T#7S
              N    "AutoProcessData".FixtureCode_A1[3]:="KeyenceSR1000Ctrl_805A1DB".sHMI.Status.CurrentCode
   END_STEP
   TRANSITION Trans293 FROM DataMove_3 TO WaitRobotScanPos4Reach   // T296
      := "AlwaysTRUE";
   END_TRANSITION
   STEP "Start 3st reading":   // S272, max time T#10S, warning time T#7S
          S1  S    "KeyenceSR1000Ctrl_805A1DB".ioAutoTrigger
   END_STEP
   TRANSITION Trans291 FROM "Start 3st reading" TO "Wait reading complete_2"   // T292
      := NOT "KeyenceSR1000Ctrl_805A1DB".sHMI.Status.Ready;
   END_TRANSITION
   STEP "Start 2st reading":   // S268, max time T#10S, warning time T#7S
          S1  S    "KeyenceSR1000Ctrl_805A1DB".ioAutoTrigger
   END_STEP
   TRANSITION Trans285 FROM "Start 2st reading" TO "Wait reading complete_1"   // T286
      := NOT "KeyenceSR1000Ctrl_805A1DB".sHMI.Status.Ready;
   END_TRANSITION
   STEP Robot2StartScan:   // S306, max time T#10S, warning time T#7S
   END_STEP
   TRANSITION Trans352 FROM Robot2StartScan TO Robot2FixtrueScanStart   // T352, jump
      := "AlwaysTRUE";
   END_TRANSITION
   STEP WaitRobotScanPos1Reach:   // S316, max time T#10S, warning time T#7S
   END_STEP
   TRANSITION Trans608 FROM WaitRobotScanPos1Reach TO "Check reader Ready"   // T608
      := "KukaRobot1_CtrlDB".sROBtoPLC.User.Cycle.DO226_ScanPos1Reach;
   END_TRANSITION
   STEP WaitRobotScanPos7Reach:   // S340, max time T#10S, warning time T#7S
              N    "KukaRobot1_CtrlDB".sPLCtoROB.User.Cycle.DI231_ScanPos6Complete
   END_STEP
   TRANSITION Trans620 FROM WaitRobotScanPos7Reach TO CheckRobot1ScanResult   // T615
      := "KukaRobot1_CtrlDB".sROBtoPLC.User.Cycle.DO233_ScanPoseFinish OR true;
   END_TRANSITION
   STEP CheckRobot1ScanResult:   // S317, max time T#10S, warning time T#7S
   END_STEP
   TRANSITION "Robot1AllScan Ok" FROM CheckRobot1ScanResult TO Robot2StartScan   // T609
      := "AutoProcessData".GlobalData.Robot1GripperCodeOKFlag AND "AutoProcessData".GlobalData.Fixture1CodeOKFlag;
   END_TRANSITION
   TRANSITION "Robot1AllScan NG" FROM CheckRobot1ScanResult TO Robot1ToMaintenance   // T373
      := #CheckRobot1ScanResult.T > t#2S;
   END_TRANSITION
   STEP WaitRobotScanGripPos1Reach:   // S329, max time T#10S, warning time T#7S
   END_STEP
   TRANSITION Trans607 FROM WaitRobotScanGripPos1Reach TO "Check reader Ready_10"   // T617
      := "KukaRobot1_CtrlDB".sROBtoPLC.User.Cycle.DO307_ScanPos1Reach;
   END_TRANSITION
   STEP "Check reader Ready_10":   // S331, max time T#10S, warning time T#7S
   END_STEP
   TRANSITION Trans629 FROM "Check reader Ready_10" TO "Start 10st reading"   // T618
      := "KeyenceSR1000Ctrl_804A1DB".oReady;
   END_TRANSITION
   STEP "Start 10st reading":   // S333, max time T#10S, warning time T#7S
          S1  S    "KeyenceSR1000Ctrl_804A1DB".ioAutoTrigger
   END_STEP
   TRANSITION Trans630 FROM "Start 10st reading" TO "Wait reading complete_10"   // T619
      := NOT "KeyenceSR1000Ctrl_804A1DB".sHMI.Status.Ready;
   END_TRANSITION
   STEP Robot1FixtureScan:   // S335, max time T#10S, warning time T#7S
              N    "AutoProcessControl".Fixture1Code.Robot1CodeReadReq
   END_STEP
   TRANSITION Trans631 FROM Robot1FixtureScan TO WaitRobotScanPos1Reach   // T620
      := "KukaRobot1_CtrlDB".sROBtoPLC.User.Cycle.DO225_ScanPosInside AND NOT "KukaRobot1_CtrlDB".sROBtoPLC.User.Cycle.DO305_GripScanInside;
   END_TRANSITION
   STEP "Wait reading complete_10":   // S295, max time T#10S, warning time T#7S
   END_STEP
   TRANSITION ReadOK_10 FROM "Wait reading complete_10" TO DataMove_10   // T351
      := "KeyenceSR1000Ctrl_804A1DB".sHMI.Status.Complete;
   END_TRANSITION
   STEP DataMove_10:   // S296, max time T#10S, warning time T#7S
              N    "AutoProcessData".GripperCode_R1[1]:="KeyenceSR1000Ctrl_804A1DB".sHMI.Status.CurrentCode
   END_STEP
   TRANSITION Trans313 FROM DataMove_10 TO RobotScanGripPos1Comp   // T355
      := TRUE;
   END_TRANSITION
   STEP RobotScanGripPos1Comp:   // S299, max time T#10S, warning time T#7S
              R    "KukaRobot1_CtrlDB".sPLCtoROB.User.Cycle.DI307_ScanPartFinish
              N    "KukaRobot1_CtrlDB".sPLCtoROB.User.Cycle.DI306_ScanPartComplete
   END_STEP
   TRANSITION Trans314 FROM RobotScanGripPos1Comp TO WaitRobotScanGripPos2Reach   // T359
      := NOT "KukaRobot1_CtrlDB".sROBtoPLC.User.Cycle.DO307_ScanPos1Reach;
   END_TRANSITION
   STEP WaitRobotScanGripPos2Reach:   // S304, max time T#10S, warning time T#7S
   END_STEP
   TRANSITION Trans316 FROM WaitRobotScanGripPos2Reach TO "Check reader Ready_11"   // T360
      := "KukaRobot1_CtrlDB".sROBtoPLC.User.Cycle.DO308_ScanPos2Reach;
   END_TRANSITION
   STEP "Check reader Ready_11":   // S337, max time T#10S, warning time T#7S
   END_STEP
   TRANSITION Trans632 FROM "Check reader Ready_11" TO "Start 11st reading"   // T621
      := "KeyenceSR1000Ctrl_804A1DB".oReady;
   END_TRANSITION
   STEP "Start 11st reading":   // S339, max time T#10S, warning time T#7S
          S1  S    "KeyenceSR1000Ctrl_804A1DB".ioAutoTrigger
   END_STEP
   TRANSITION Trans633 FROM "Start 11st reading" TO "Wait reading complete_11"   // T622
      := NOT "KeyenceSR1000Ctrl_804A1DB".sHMI.Status.Ready;
   END_TRANSITION
   STEP "Wait reading complete_11":   // S342, max time T#10S, warning time T#7S
   END_STEP
   TRANSITION ReadOK_11 FROM "Wait reading complete_11" TO DataMove_11   // T361
      := "KeyenceSR1000Ctrl_804A1DB".sHMI.Status.Complete;
   END_TRANSITION
   STEP DataMove_11:   // S343, max time T#10S, warning time T#7S
              N    "AutoProcessData".GripperCode_R1[2]:="KeyenceSR1000Ctrl_804A1DB".sHMI.Status.CurrentCode
   END_STEP
   TRANSITION Trans318 FROM DataMove_11 TO RobotScanGripPos2Comp   // T364
      := TRUE;
   END_TRANSITION
   STEP RobotScanGripPos2Comp:   // S345, max time T#10S, warning time T#7S
              R    "KukaRobot1_CtrlDB".sPLCtoROB.User.Cycle.DI307_ScanPartFinish
              N    "KukaRobot1_CtrlDB".sPLCtoROB.User.Cycle.DI306_ScanPartComplete
   END_STEP
   TRANSITION Trans319 FROM RobotScanGripPos2Comp TO WaitRobotScanGripPos3Reach   // T367
      := NOT "KukaRobot1_CtrlDB".sROBtoPLC.User.Cycle.DO308_ScanPos2Reach;
   END_TRANSITION
   STEP WaitRobotScanGripPos3Reach:   // S346, max time T#10S, warning time T#7S
   END_STEP
   TRANSITION Trans320 FROM WaitRobotScanGripPos3Reach TO "Check reader Ready_12"   // T368
      := "KukaRobot1_CtrlDB".sROBtoPLC.User.Cycle.DO309_ScanPos3Reach;
   END_TRANSITION
   STEP "Check reader Ready_12":   // S347, max time T#10S, warning time T#7S
   END_STEP
   TRANSITION Trans634 FROM "Check reader Ready_12" TO "Start 11st reading_1"   // T623
      := "KeyenceSR1000Ctrl_804A1DB".oReady;
   END_TRANSITION
   STEP "Start 11st reading_1":   // S348, max time T#10S, warning time T#7S
          S1  S    "KeyenceSR1000Ctrl_804A1DB".ioAutoTrigger
   END_STEP
   TRANSITION Trans635 FROM "Start 11st reading_1" TO "Wait reading complete_12"   // T624
      := NOT "KeyenceSR1000Ctrl_804A1DB".sHMI.Status.Ready;
   END_TRANSITION
   STEP "Wait reading complete_12":   // S350, max time T#10S, warning time T#7S
   END_STEP
   TRANSITION ReadOK_12 FROM "Wait reading complete_12" TO DataMove_12   // T369
      := "KeyenceSR1000Ctrl_804A1DB".sHMI.Status.Complete;
   END_TRANSITION
   STEP DataMove_12:   // S351, max time T#10S, warning time T#7S
              N    "AutoProcessData".GripperCode_R1[3]:="KeyenceSR1000Ctrl_804A1DB".sHMI.Status.CurrentCode
   END_STEP
   TRANSITION Trans322 FROM DataMove_12 TO RobotScanGripPos3Comp   // T372
      := TRUE;
   END_TRANSITION
   STEP RobotScanGripPos3Comp:   // S353, max time T#10S, warning time T#7S
              R    "KukaRobot1_CtrlDB".sPLCtoROB.User.Cycle.DI307_ScanPartFinish
              N    "KukaRobot1_CtrlDB".sPLCtoROB.User.Cycle.DI306_ScanPartComplete
   END_STEP
   TRANSITION Trans323 FROM RobotScanGripPos3Comp TO WaitRobotScanGripPos4Reach   // T375
      := NOT "KukaRobot1_CtrlDB".sROBtoPLC.User.Cycle.DO309_ScanPos3Reach;
   END_TRANSITION
   STEP WaitRobotScanGripPos4Reach:   // S354, max time T#10S, warning time T#7S
   END_STEP
   TRANSITION Trans324 FROM WaitRobotScanGripPos4Reach TO "Check reader Ready_13"   // T376
      := "KukaRobot1_CtrlDB".sROBtoPLC.User.Cycle.DO310_ScanPos4Reach;
   END_TRANSITION
   STEP "Check reader Ready_13":   // S355, max time T#10S, warning time T#7S
   END_STEP
   TRANSITION Trans636 FROM "Check reader Ready_13" TO "Start 11st reading_2"   // T625
      := "KeyenceSR1000Ctrl_804A1DB".oReady;
   END_TRANSITION
   STEP "Start 11st reading_2":   // S356, max time T#10S, warning time T#7S
          S1  S    "KeyenceSR1000Ctrl_804A1DB".ioAutoTrigger
   END_STEP
   TRANSITION Trans637 FROM "Start 11st reading_2" TO "Wait reading complete_13"   // T626
      := NOT "KeyenceSR1000Ctrl_804A1DB".sHMI.Status.Ready;
   END_TRANSITION
   STEP "Wait reading complete_13":   // S358, max time T#10S, warning time T#7S
   END_STEP
   TRANSITION ReadOK_13 FROM "Wait reading complete_13" TO DataMove_13   // T377
      := "KeyenceSR1000Ctrl_804A1DB".sHMI.Status.Complete;
   END_TRANSITION
   STEP DataMove_13:   // S359, max time T#10S, warning time T#7S
              N    "AutoProcessData".GripperCode_R1[4]:="KeyenceSR1000Ctrl_804A1DB".sHMI.Status.CurrentCode
   END_STEP
   TRANSITION Trans327 FROM DataMove_13 TO RobotScanGripPos4Comp   // T380
      := TRUE;
   END_TRANSITION
   STEP RobotScanGripPos4Comp:   // S361, max time T#10S, warning time T#7S
              N    "KukaRobot1_CtrlDB".sPLCtoROB.User.Cycle.DI307_ScanPartFinish
              N    "KukaRobot1_CtrlDB".sPLCtoROB.User.Cycle.DI306_ScanPartComplete
   END_STEP
   TRANSITION Trans328 FROM RobotScanGripPos4Comp TO Robot1FixtureScan   // T383
      := "KukaRobot1_CtrlDB".sROBtoPLC.User.Cycle.DO306_GripScanFinish;
   END_TRANSITION
   STEP WaitServoStop:   // S422, max time T#10S, warning time T#7S
   END_STEP
   TRANSITION Trans422 FROM WaitServoStop TO "Check reader Ready_4"   // T422
      := "iC-GlueServoHomePos";
   END_TRANSITION

   // sequencer 4: S600-S699工件放行 / S300-S399 Robot2 FixtureCode reading
   STEP Robot2FixtrueScanStart:   // S300, max time T#10S, warning time T#7S
              R    "KukaRobot2_CtrlDB".sPLCtoROB.User.Cycle.DI307_ScanPartFinish
              R    "KukaRobot2_CtrlDB".sPLCtoROB.User.Cycle.DI306_ScanPartComplete
              N    "AutoProcessData".GripperCode_R2[1]:=''
              N    "AutoProcessData".GripperCode_R2[2]:=''
              N    "AutoProcessData".GripperCode_R2[3]:=''
              N    "AutoProcessData".GripperCode_R2[4]:=''
   END_STEP
   TRANSITION Trans302 FROM Robot2FixtrueScanStart TO Robot2CheckScanStatus   // T300
      := ("KukaRobot1_CtrlDB".sROBtoPLC.Sys.SO.IN_HOME OR "KukaRobot1_CtrlDB".sROBtoPLC.User.Cycle.DO298_MaintainFinish) AND (NOT "KukaRobot1_CtrlDB".sROBtoPLC.User.Cycle.DO225_ScanPosInside OR "KukaRobot1_CtrlDB".sROBtoPLC.Sys.SO.IN_HOME);
   END_TRANSITION
   STEP "Check reader Ready_14":   // S341, max time T#10S, warning time T#7S
   END_STEP
   TRANSITION Trans638 FROM "Check reader Ready_14" TO "Start 10st reading_1"   // T627
      := "KeyenceSR1000Ctrl_806A1DB".oReady;
   END_TRANSITION
   STEP Robot2CheckScanResult:   // S149, max time T#10S, warning time T#7S
   END_STEP
   TRANSITION R2ScanOk FROM Robot2CheckScanResult TO Robot3StartToScan   // T149
      := "AutoProcessData".GlobalData.Robot2GripperCodeOKFlag;
   END_TRANSITION
   TRANSITION R2ScanNG FROM Robot2CheckScanResult TO Robot2StartToMaintenanc   // T675
      := NOT "AutoProcessData".GlobalData.Robot2GripperCodeOKFlag AND (#Robot2CheckScanResult.T > t#2S);
   END_TRANSITION
   STEP Robot3StartToScan:   // S365, max time T#10S, warning time T#7S
   END_STEP
   TRANSITION Trans674 FROM Robot3StartToScan TO Robot3FixtrueScanStart   // T674, jump
      := NOT "KukaRobot2_CtrlDB".sROBtoPLC.User.Cycle.DO297_MaintainInside;
   END_TRANSITION
   STEP Robot2StartToMaintenanc:   // S366, max time T#10S, warning time T#7S
   END_STEP
   TRANSITION Trans678 FROM Robot2StartToMaintenanc TO Step720   // T676, jump
      := TRUE;
   END_TRANSITION
   STEP "Start 10st reading_1":   // S344, max time T#10S, warning time T#7S
          S1  S    "KeyenceSR1000Ctrl_806A1DB".ioAutoTrigger
   END_STEP
   TRANSITION Trans642 FROM "Start 10st reading_1" TO "Wait reading complete_14"   // T628
      := NOT "KeyenceSR1000Ctrl_806A1DB".sHMI.Status.Ready;
   END_TRANSITION
   STEP "Wait reading complete_14":   // S297, max time T#10S, warning time T#7S
   END_STEP
   TRANSITION ReadOK_14 FROM "Wait reading complete_14" TO DataMove_14   // T354
      := "KeyenceSR1000Ctrl_806A1DB".sHMI.Status.Complete;
   END_TRANSITION
   STEP DataMove_14:   // S303, max time T#10S, warning time T#7S
              N    "AutoProcessData".GripperCode_R2[1]:="KeyenceSR1000Ctrl_806A1DB".sHMI.Status.CurrentCode
   END_STEP
   TRANSITION Trans315 FROM DataMove_14 TO RobotScanGripPos1Comp_1   // T356
      := "AlwaysTRUE";
   END_TRANSITION
   STEP RobotScanGripPos1Comp_1:   // S305, max time T#10S, warning time T#7S
              R    "KukaRobot2_CtrlDB".sPLCtoROB.User.Cycle.DI307_ScanPartFinish
              N    "KukaRobot2_CtrlDB".sPLCtoROB.User.Cycle.DI306_ScanPartComplete
   END_STEP
   TRANSITION Trans317 FROM RobotScanGripPos1Comp_1 TO WaitRobotScanGripPos2Reach_1   // T362
      := NOT "KukaRobot2_CtrlDB".sROBtoPLC.User.Cycle.DO307_ScanPos1Reach;
   END_TRANSITION
   STEP WaitRobotScanGripPos2Reach_1:   // S307, max time T#10S, warning time T#7S
   END_STEP
   TRANSITION Trans321 FROM WaitRobotScanGripPos2Reach_1 TO "Check reader Ready_15"   // T363
      := "KukaRobot2_CtrlDB".sROBtoPLC.User.Cycle.DO308_ScanPos2Reach;
   END_TRANSITION
   STEP "Check reader Ready_15":   // S352, max time T#10S, warning time T#7S
   END_STEP
   TRANSITION Trans652 FROM "Check reader Ready_15" TO "Start 11st reading_3"   // T630
      := "KeyenceSR1000Ctrl_806A1DB".oReady;
   END_TRANSITION
   STEP "Start 11st reading_3":   // S357, max time T#10S, warning time T#7S
          S1  S    "KeyenceSR1000Ctrl_806A1DB".ioAutoTrigger
   END_STEP
   TRANSITION Trans653 FROM "Start 11st reading_3" TO "Wait reading complete_15"   // T631
      := NOT "KeyenceSR1000Ctrl_806A1DB".sHMI.Status.Ready;
   END_TRANSITION
   STEP "Wait reading complete_15":   // S360, max time T#10S, warning time T#7S
   END_STEP
   TRANSITION ReadOK_15 FROM "Wait reading complete_15" TO DataMove_15   // T365
      := "KeyenceSR1000Ctrl_806A1DB".sHMI.Status.Complete;
   END_TRANSITION
   STEP DataMove_15:   // S362, max time T#10S, warning time T#7S
              N    "AutoProcessData".GripperCode_R2[2]:="KeyenceSR1000Ctrl_806A1DB".sHMI.Status.CurrentCode
   END_STEP
   TRANSITION Trans326 FROM DataMove_15 TO RobotScanGripPos2Comp_1   // T366
      := "AlwaysTRUE";
   END_TRANSITION
   STEP RobotScanGripPos2Comp_1:   // S371, max time T#10S, warning time T#7S
              R    "KukaRobot2_CtrlDB".sPLCtoROB.User.Cycle.DI307_ScanPartFinish
              N    "KukaRobot2_CtrlDB".sPLCtoROB.User.Cycle.DI306_ScanPartComplete
   END_STEP
   TRANSITION Trans329 FROM RobotScanGripPos2Comp_1 TO WaitRobotScanGripPos3Reach_1   // T370
      := NOT "KukaRobot2_CtrlDB".sROBtoPLC.User.Cycle.DO308_ScanPos2Reach;
   END_TRANSITION
   STEP WaitRobotScanGripPos3Reach_1:   // S372, max time T#10S, warning time T#7S
   END_STEP
   TRANSITION Trans330 FROM WaitRobotScanGripPos3Reach_1 TO "Check reader Ready_16"   // T371
      := "KukaRobot2_CtrlDB".sROBtoPLC.User.Cycle.DO309_ScanPos3Reach;
   END_TRANSITION
   STEP "Check reader Ready_16":   // S373, max time T#10S, warning time T#7S
   END_STEP
   TRANSITION Trans673 FROM "Check reader Ready_16" TO "Start 11st reading_4"   // T632
      := "KeyenceSR1000Ctrl_806A1DB".oReady;
   END_TRANSITION
   STEP "Start 11st reading_4":   // S374, max time T#10S, warning time T#7S
          S1  S    "KeyenceSR1000Ctrl_806A1DB".ioAutoTrigger
   END_STEP
   TRANSITION Trans675 FROM "Start 11st reading_4" TO "Wait reading complete_16"   // T633
      := NOT "KeyenceSR1000Ctrl_806A1DB".sHMI.Status.Ready;
   END_TRANSITION
   STEP "Wait reading complete_16":   // S375, max time T#10S, warning time T#7S
   END_STEP
   TRANSITION ReadOK_16 FROM "Wait reading complete_16" TO DataMove_16   // T374
      := "KeyenceSR1000Ctrl_806A1DB".sHMI.Status.Complete;
   END_TRANSITION
   STEP DataMove_16:   // S376, max time T#10S, warning time T#7S
              N    "AutoProcessData".GripperCode_R2[3]:="KeyenceSR1000Ctrl_806A1DB".sHMI.Status.CurrentCode
   END_STEP
   TRANSITION Trans331 FROM DataMove_16 TO RobotScanGripPos3Comp_1   // T378
      := "AlwaysTRUE";
   END_TRANSITION
   STEP RobotScanGripPos3Comp_1:   // S378, max time T#10S, warning time T#7S
              R    "KukaRobot2_CtrlDB".sPLCtoROB.User.Cycle.DI307_ScanPartFinish
              N    "KukaRobot2_CtrlDB".sPLCtoROB.User.Cycle.DI306_ScanPartComplete
   END_STEP
   TRANSITION Trans332 FROM RobotScanGripPos3Comp_1 TO WaitRobotScanGripPos4Reach_1   // T379
      := NOT "KukaRobot2_CtrlDB".sROBtoPLC.User.Cycle.DO309_ScanPos3Reach;
   END_TRANSITION
   STEP WaitRobotScanGripPos4Reach_1:   // S383, max time T#10S, warning time T#7S
   END_STEP
   TRANSITION Trans333 FROM WaitRobotScanGripPos4Reach_1 TO "Check reader Ready_17"   // T381
      := "KukaRobot2_CtrlDB".sROBtoPLC.User.Cycle.DO310_ScanPos4Reach;
   END_TRANSITION
   STEP "Check reader Ready_17":   // S385, max time T#10S, warning time T#7S
   END_STEP
   TRANSITION Trans676 FROM "Check reader Ready_17" TO "Start 11st reading_5"   // T635
      := "KeyenceSR1000Ctrl_806A1DB".oReady;
   END_TRANSITION
   STEP "Start 11st reading_5":   // S386, max time T#10S, warning time T#7S
          S1  S    "KeyenceSR1000Ctrl_806A1DB".ioAutoTrigger
   END_STEP
   TRANSITION Trans677 FROM "Start 11st reading_5" TO "Wait reading complete_17"   // T638
      := NOT "KeyenceSR1000Ctrl_806A1DB".sHMI.Status.Ready;
   END_TRANSITION
   STEP "Wait reading complete_17":   // S388, max time T#10S, warning time T#7S
   END_STEP
   TRANSITION ReadOK_17 FROM "Wait reading complete_17" TO DataMove_17   // T382
      := "KeyenceSR1000Ctrl_806A1DB".sHMI.Status.Complete;
   END_TRANSITION
   STEP DataMove_17:   // S389, max time T#10S, warning time T#7S
              N    "AutoProcessData".GripperCode_R2[4]:="KeyenceSR1000Ctrl_806A1DB".sHMI.Status.CurrentCode
   END_STEP
   TRANSITION Trans334 FROM DataMove_17 TO RobotScanGripPos4Comp_1   // T384
      := "AlwaysTRUE";
   END_TRANSITION
   STEP RobotScanGripPos4Comp_1:   // S391, max time T#10S, warning time T#7S
              N    "KukaRobot2_CtrlDB".sPLCtoROB.User.Cycle.DI307_ScanPartFinish
              N    "KukaRobot2_CtrlDB".sPLCtoROB.User.Cycle.DI306_ScanPartComplete
   END_STEP
   TRANSITION Trans335 FROM RobotScanGripPos4Comp_1 TO Robot2CheckScanResult   // T385
      := "KukaRobot2_CtrlDB".sROBtoPLC.User.Cycle.DO306_GripScanFinish;
   END_TRANSITION
   STEP StartRobotScanGripperCode:   // S363, max time T#10S, warning time T#7S
              N    "AutoProcessControl".Robot_2.GripScanRequest
   END_STEP
   TRANSITION Trans684 FROM StartRobotScanGripperCode TO RobotScanGripperReachPos1   // T616
      := "KukaRobot2_CtrlDB".sROBtoPLC.User.Cycle.DO305_GripScanInside AND NOT "KukaRobot2_CtrlDB".sROBtoPLC.User.Cycle.DO306_GripScanFinish;
   END_TRANSITION
   STEP RobotScanGripperReachPos1:   // S364, max time T#10S, warning time T#7S
   END_STEP
   TRANSITION Trans685 FROM RobotScanGripperReachPos1 TO "Check reader Ready_14"   // T673
      := "KukaRobot2_CtrlDB".sROBtoPLC.User.Cycle.DO307_ScanPos1Reach;
   END_TRANSITION
   STEP Robot2CheckScanStatus:   // S410, max time T#10S, warning time T#7S
   END_STEP
   TRANSITION "317GripScanng" FROM Robot2CheckScanStatus TO StartRobotScanGripperCode   // T317
      := NOT "AutoProcessData".GlobalData.Robot2GripperCodeOKFlag;
   END_TRANSITION
   TRANSITION "319GripScanOK" FROM Robot2CheckScanStatus TO Robot2CheckScanResult   // T319
      := "AutoProcessData".GlobalData.Robot2GripperCodeOKFlag;
   END_TRANSITION

   // sequencer 5: S400-S499 Robot3 FixtureCode reading
   STEP Robot3FixtrueScanStart:   // S400, max time T#10S, warning time T#7S
              N    "AutoProcessData".GripperCode_R3[1]:=''
              N    "AutoProcessData".GripperCode_R3[2]:=''
              N    "AutoProcessData".GripperCode_R3[3]:=''
              N    "AutoProcessData".GripperCode_R3[4]:=''
              N    "AutoProcessData".FixtureCode_A2[1]:=''
              N    "AutoProcessData".FixtureCode_A2[2]:=''
              N    "AutoProcessData".FixtureCode_A2[3]:=''
              N    "AutoProcessData".FixtureCode_A2[4]:=''
              N    "AutoProcessData".FixtureCode_A2[5]:=''
              N    "AutoProcessData".FixtureCode_A2[6]:=''
              N    "AutoProcessData".FixtureCode_A2[7]:=''
              N    "AutoProcessData".FixtureCode_A2[8]:=''
   END_STEP
   TRANSITION Trans400 FROM Robot3FixtrueScanStart TO Robot3CheckScanStatus   // T400
      := NOT "KukaRobot2_CtrlDB".sROBtoPLC.User.Cycle.DO297_MaintainInside;
   END_TRANSITION
   STEP AllScanFinish:   // S408, max time T#10S, warning time T#7S
   END_STEP
   TRANSITION Trans403 FROM AllScanFinish TO ProcessStart   // T403, jump
      := "AutoProcessData".GlobalData.Table1CodeOKFlag AND "AutoProcessData".GlobalData.Table2CodeOKFlag AND "AutoProcessData".GlobalData.Robot1GripperCodeOKFlag AND "AutoProcessData".GlobalData.Robot2GripperCodeOKFlag AND "AutoProcessData".GlobalData.Robot3GripperCodeOKFlag AND "AutoProcessData".GlobalData.Fixture1CodeOKFlag AND "AutoProcessData".GlobalData.Fixture2CodeOKFlag AND "ST10_RecipeDB".Recipe.Equal AND NOT "ChangeOver_DB".Global.ScanFixtureFlag AND NOT "ChangeOver_DB".Global.ChangeOverRequest;
   END_TRANSITION
   TRANSITION Trans420 FROM AllScanFinish TO ProcessStart   // T420, jump
      := ("ChangeOver_DB".Global.ChangeOverRequest OR "ChangeOver_DB".Global.ChangeOverSelected) AND NOT "ChangeOver_DB".Global.ChangeOverSelected;
   END_TRANSITION
   STEP DataMove_7:   // S279, max time T#10S, warning time T#7S
              N    "AutoProcessData".FixtureCode_A2[2]:="KeyenceSR1000Ctrl_807A1DB".sHMI.Status.CurrentCode
   END_STEP
   TRANSITION Trans336 FROM DataMove_7 TO WaitRobotScanPos3Reach_1   // T312
      := "AlwaysTRUE";
   END_TRANSITION
   STEP Robot3StartToMaintenance:   // S409, max time T#10S, warning time T#7S
   END_STEP
   TRANSITION Trans405 FROM Robot3StartToMaintenance TO Step712   // T405, jump
      := TRUE;
   END_TRANSITION
   STEP DataMove_8:   // S284, max time T#10S, warning time T#7S
              N    "AutoProcessData".FixtureCode_A2[1]:="KeyenceSR1000Ctrl_807A1DB".sHMI.Status.CurrentCode
   END_STEP
   TRANSITION Trans290 FROM DataMove_8 TO WaitRobotScanPos2Reach_1   // T301
      := "AlwaysTRUE";
   END_TRANSITION
   STEP RequestRobotScanFixture:   // S312, max time T#10S, warning time T#7S
              N    "AutoProcessControl".Fixture2Code.Robot3CodeReadReq
   END_STEP
   TRANSITION Trans609 FROM RequestRobotScanFixture TO WaitRobotScanPos1Reach_3   // T634
      := "KukaRobot3_CtrlDB".sROBtoPLC.User.Cycle.DO225_ScanPosInside;
   END_TRANSITION
   STEP "Start 1st reading_1":   // S289, max time T#10S, warning time T#7S
          S1  S    "KeyenceSR1000Ctrl_807A1DB".ioAutoTrigger
   END_STEP
   TRANSITION Trans284 FROM "Start 1st reading_1" TO "Wait reading complete_6"   // T283
      := NOT "KeyenceSR1000Ctrl_807A1DB".sHMI.Status.Ready;
   END_TRANSITION
   STEP "Check reader Ready_6":   // S290, max time T#10S, warning time T#7S
   END_STEP
   TRANSITION Trans280 FROM "Check reader Ready_6" TO "Start 1st reading_1"   // T297
      := "KeyenceSR1000Ctrl_807A1DB".sHMI.Status.Ready;
   END_TRANSITION
   STEP "Wait reading complete_6":   // S291, max time T#10S, warning time T#7S
   END_STEP
   TRANSITION ReadOK_8 FROM "Wait reading complete_6" TO DataMove_8   // T285
      := "KeyenceSR1000Ctrl_807A1DB".sHMI.Status.Complete;
   END_TRANSITION
   STEP WaitRobotScanPos1Reach_2:   // S367, max time T#10S, warning time T#7S
              N    "KukaRobot3_CtrlDB".sPLCtoROB.User.Cycle.DI230_ScanPos5Complete
   END_STEP
   TRANSITION Trans618 FROM WaitRobotScanPos1Reach_2 TO "Check reader Ready_23"   // T636
      := "KukaRobot3_CtrlDB".sROBtoPLC.User.Cycle.DO233_ScanPoseFinish;
   END_TRANSITION
   STEP WaitRobotScanPos5Reach_1:   // S368, max time T#10S, warning time T#7S
              N    "KukaRobot3_CtrlDB".sPLCtoROB.User.Cycle.DI229_ScanPos4Complete
   END_STEP
   TRANSITION Trans619 FROM WaitRobotScanPos5Reach_1 TO "Check reader Ready_7"   // T637
      := "KukaRobot3_CtrlDB".sROBtoPLC.User.Cycle.DO230_ScanPos5Reach;
   END_TRANSITION
   STEP WaitRobotScanPos2Reach_1:   // S369, max time T#10S, warning time T#7S
              N    "KukaRobot3_CtrlDB".sPLCtoROB.User.Cycle.DI226_ScanPos1Complete
   END_STEP
   TRANSITION Trans623 FROM WaitRobotScanPos2Reach_1 TO "Check reader Ready_18"   // T641
      := "KukaRobot3_CtrlDB".sROBtoPLC.User.Cycle.DO227_ScanPos2Reach;
   END_TRANSITION
   STEP WaitRobotScanPos4Reach_1:   // S370, max time T#10S, warning time T#7S
              N    "KukaRobot3_CtrlDB".sPLCtoROB.User.Cycle.DI228_ScanPos3Complete
   END_STEP
   TRANSITION Trans621 FROM WaitRobotScanPos4Reach_1 TO "Check reader Ready_8"   // T639
      := "KukaRobot3_CtrlDB".sROBtoPLC.User.Cycle.DO229_ScanPos4Reach;
   END_TRANSITION
   STEP "Start 5st reading_1":   // S292, max time T#10S, warning time T#7S
          S1  S    "KeyenceSR1000Ctrl_807A1DB".ioAutoTrigger
   END_STEP
   TRANSITION Trans307 FROM "Start 5st reading_1" TO "Wait reading complete_7"   // T314
      := NOT "KeyenceSR1000Ctrl_807A1DB".sHMI.Status.Ready;
   END_TRANSITION
   STEP "Check reader Ready_7":   // S293, max time T#10S, warning time T#7S
   END_STEP
   TRANSITION Trans308 FROM "Check reader Ready_7" TO "Start 5st reading_1"   // T327
      := "KeyenceSR1000Ctrl_807A1DB".sHMI.Status.Ready;
   END_TRANSITION
   STEP "Wait reading complete_7":   // S294, max time T#10S, warning time T#7S
   END_STEP
   TRANSITION ReadOK_18 FROM "Wait reading complete_7" TO DataMove_9   // T316
      := "KeyenceSR1000Ctrl_807A1DB".sHMI.Status.Complete;
   END_TRANSITION
   STEP "Wait reading complete_8":   // S301, max time T#10S, warning time T#7S
   END_STEP
   TRANSITION ReadOK_9 FROM "Wait reading complete_8" TO DataMove_18   // T302
      := "KeyenceSR1000Ctrl_807A1DB".sHMI.Status.Complete;
   END_TRANSITION
   STEP "Check reader Ready_8":   // S302, max time T#10S, warning time T#7S
   END_STEP
   TRANSITION Trans298 FROM "Check reader Ready_8" TO "Start 4st reading_1"   // T308
      := "KeyenceSR1000Ctrl_807A1DB".sHMI.Status.Ready;
   END_TRANSITION
   STEP DataMove_9:   // S309, max time T#10S, warning time T#7S
              N    "AutoProcessData".FixtureCode_A2[5]:="KeyenceSR1000Ctrl_807A1DB".sHMI.Status.CurrentCode
   END_STEP
   TRANSITION Trans303 FROM DataMove_9 TO WaitRobotScanPos1Reach_2   // T324
      := "AlwaysTRUE";
   END_TRANSITION
   STEP DataMove_18:   // S310, max time T#10S, warning time T#7S
              N    "AutoProcessData".FixtureCode_A2[4]:="KeyenceSR1000Ctrl_807A1DB".sHMI.Status.CurrentCode
   END_STEP
   TRANSITION Trans309 FROM DataMove_18 TO WaitRobotScanPos5Reach_1   // T309
      := "AlwaysTRUE";
   END_TRANSITION
   STEP "Start 4st reading_1":   // S313, max time T#10S, warning time T#7S
          S1  S    "KeyenceSR1000Ctrl_807A1DB".ioAutoTrigger
   END_STEP
   TRANSITION Trans310 FROM "Start 4st reading_1" TO "Wait reading complete_8"   // T304
      := NOT "KeyenceSR1000Ctrl_807A1DB".sHMI.Status.Ready;
   END_TRANSITION
   STEP "Check reader Ready_9":   // S314, max time T#10S, warning time T#7S
   END_STEP
   TRANSITION Trans311 FROM "Check reader Ready_9" TO "Start 3st reading_1"   // T305
      := "KeyenceSR1000Ctrl_807A1DB".sHMI.Status.Ready;
   END_TRANSITION
   STEP "Wait reading complete_9":   // S315, max time T#10S, warning time T#7S
   END_STEP
   TRANSITION ReadOK_19 FROM "Wait reading complete_9" TO DataMove_19   // T311
      := "KeyenceSR1000Ctrl_807A1DB".sHMI.Status.Complete;
   END_TRANSITION
   STEP WaitRobotScanPos3Reach_1:   // S377, max time T#10S, warning time T#7S
              N    "KukaRobot3_CtrlDB".sPLCtoROB.User.Cycle.DI227_ScanPos2Complete
   END_STEP
   TRANSITION Trans622 FROM WaitRobotScanPos3Reach_1 TO "Check reader Ready_9"   // T640
      := "KukaRobot3_CtrlDB".sROBtoPLC.User.Cycle.DO228_ScanPos3Reach;
   END_TRANSITION
   STEP "Check reader Ready_18":   // S318, max time T#10S, warning time T#7S
   END_STEP
   TRANSITION Trans288 FROM "Check reader Ready_18" TO "Start 2st reading_1"   // T291
      := "KeyenceSR1000Ctrl_807A1DB".sHMI.Status.Ready;
   END_TRANSITION
   STEP "Wait reading complete_18":   // S319, max time T#10S, warning time T#7S
   END_STEP
   TRANSITION ReadOK_7 FROM "Wait reading complete_18" TO DataMove_7   // T288
      := "KeyenceSR1000Ctrl_807A1DB".sHMI.Status.Complete;
   END_TRANSITION
   STEP DataMove_19:   // S320, max time T#10S, warning time T#7S
              N    "AutoProcessData".FixtureCode_A2[3]:="KeyenceSR1000Ctrl_807A1DB".sHMI.Status.CurrentCode
   END_STEP
   TRANSITION Trans312 FROM DataMove_19 TO WaitRobotScanPos4Reach_1   // T310
      := "AlwaysTRUE";
   END_TRANSITION
   STEP "Start 3st reading_1":   // S321, max time T#10S, warning time T#7S
          S1  S    "KeyenceSR1000Ctrl_807A1DB".ioAutoTrigger
   END_STEP
   TRANSITION Trans294 FROM "Start 3st reading_1" TO "Wait reading complete_9"   // T303
      := NOT "KeyenceSR1000Ctrl_807A1DB".sHMI.Status.Ready;
   END_TRANSITION
   STEP "Start 2st reading_1":   // S322, max time T#10S, warning time T#7S
          S1  S    "KeyenceSR1000Ctrl_807A1DB".ioAutoTrigger
   END_STEP
   TRANSITION Trans289 FROM "Start 2st reading_1" TO "Wait reading complete_18"   // T294
      := NOT "KeyenceSR1000Ctrl_807A1DB".sHMI.Status.Ready;
   END_TRANSITION
   STEP Robot3CheckScanResult:   // S323, max time T#10S, warning time T#7S
   END_STEP
   TRANSITION R3ScanOk FROM Robot3CheckScanResult TO AllScanFinish   // T357
      := "AutoProcessData".GlobalData.Fixture2CodeOKFlag AND "AutoProcessData".GlobalData.Robot3GripperCodeOKFlag;
   END_TRANSITION
   TRANSITION R3ScanNG FROM Robot3CheckScanResult TO Robot3StartToMaintenance   // T404
      := #Robot3CheckScanResult.T > t#2S;
   END_TRANSITION
   STEP WaitRobotScanPos1Reach_3:   // S324, max time T#10S, warning time T#7S
   END_STEP
   TRANSITION Trans610 FROM WaitRobotScanPos1Reach_3 TO "Check reader Ready_6"   // T642
      := "KukaRobot3_CtrlDB".sROBtoPLC.User.Cycle.DO226_ScanPos1Reach;
   END_TRANSITION
   STEP RequestRobotScan_1:   // S379, max time T#10S, warning time T#7S
              N    "AutoProcessControl".Robot_3.GripScanRequest
   END_STEP
   TRANSITION Trans639 FROM RequestRobotScan_1 TO WaitRobotScanGripPos1Reach_1   // T643
      := NOT "KukaRobot3_CtrlDB".sROBtoPLC.User.Cycle.DO225_ScanPosInside AND "KukaRobot3_CtrlDB".sROBtoPLC.User.Cycle.DO305_GripScanInside;
   END_TRANSITION
   STEP WaitRobotScanGripPos1Reach_1:   // S380, max time T#10S, warning time T#7S
   END_STEP
   TRANSITION Trans640 FROM WaitRobotScanGripPos1Reach_1 TO "Check reader Ready_19"   // T644
      := "KukaRobot3_CtrlDB".sROBtoPLC.User.Cycle.DO307_ScanPos1Reach;
   END_TRANSITION
   STEP "Check reader Ready_19":   // S381, max time T#10S, warning time T#7S
   END_STEP
   TRANSITION Trans641 FROM "Check reader Ready_19" TO "Start 10st reading_2"   // T645
      := "KeyenceSR1000Ctrl_803A1DB".oReady;
   END_TRANSITION
   STEP "Start 10st reading_2":   // S382, max time T#10S, warning time T#7S
          S1  S    "KeyenceSR1000Ctrl_803A1DB".ioAutoTrigger
   END_STEP
   TRANSITION Trans643 FROM "Start 10st reading_2" TO "Wait reading complete_19"   // T646
      := NOT "KeyenceSR1000Ctrl_803A1DB".sHMI.Status.Ready;
   END_TRANSITION
   STEP "Wait reading complete_19":   // S325, max time T#10S, warning time T#7S
   END_STEP
   TRANSITION ReadOK_20 FROM "Wait reading complete_19" TO DataMove_20   // T386
      := "KeyenceSR1000Ctrl_803A1DB".sHMI.Status.Complete;
   END_TRANSITION
   STEP DataMove_20:   // S326, max time T#10S, warning time T#7S
              N    "AutoProcessData".GripperCode_R3[1]:="KeyenceSR1000Ctrl_803A1DB".sHMI.Status.CurrentCode
   END_STEP
   TRANSITION Trans337 FROM DataMove_20 TO RobotScanGripPos1Comp_2   // T387
      := "AlwaysTRUE";
   END_TRANSITION
   STEP RobotScanGripPos1Comp_2:   // S327, max time T#10S, warning time T#7S
              R    "KukaRobot3_CtrlDB".sPLCtoROB.User.Cycle.DI307_ScanPartFinish
              N    "KukaRobot3_CtrlDB".sPLCtoROB.User.Cycle.DI306_ScanPartComplete
   END_STEP
   TRANSITION Trans338 FROM RobotScanGripPos1Comp_2 TO WaitRobotScanGripPos2Reach_2   // T388
      := NOT "KukaRobot3_CtrlDB".sROBtoPLC.User.Cycle.DO307_ScanPos1Reach;
   END_TRANSITION
   STEP WaitRobotScanGripPos2Reach_2:   // S328, max time T#10S, warning time T#7S
   END_STEP
   TRANSITION Trans339 FROM WaitRobotScanGripPos2Reach_2 TO "Check reader Ready_20"   // T389
      := "KukaRobot3_CtrlDB".sROBtoPLC.User.Cycle.DO308_ScanPos2Reach;
   END_TRANSITION
   STEP "Check reader Ready_20":   // S384, max time T#10S, warning time T#7S
   END_STEP
   TRANSITION Trans644 FROM "Check reader Ready_20" TO "Start 11st reading_6"   // T647
      := "KeyenceSR1000Ctrl_803A1DB".oReady;
   END_TRANSITION
   STEP "Start 11st reading_6":   // S387, max time T#10S, warning time T#7S
          S1  S    "KeyenceSR1000Ctrl_803A1DB".ioAutoTrigger
   END_STEP
   TRANSITION Trans645 FROM "Start 11st reading_6" TO "Wait reading complete_20"   // T648
      := NOT "KeyenceSR1000Ctrl_803A1DB".sHMI.Status.Ready;
   END_TRANSITION
   STEP "Wait reading complete_20":   // S390, max time T#10S, warning time T#7S
   END_STEP
   TRANSITION ReadOK_21 FROM "Wait reading complete_20" TO DataMove_21   // T390
      := "KeyenceSR1000Ctrl_803A1DB".sHMI.Status.Complete;
   END_TRANSITION
   STEP DataMove_21:   // S392, max time T#10S, warning time T#7S
              N    "AutoProcessData".GripperCode_R3[2]:="KeyenceSR1000Ctrl_803A1DB".sHMI.Status.CurrentCode
   END_STEP
   TRANSITION Trans340 FROM DataMove_21 TO RobotScanGripPos2Comp_2   // T391
      := "AlwaysTRUE";
   END_TRANSITION
   STEP RobotScanGripPos2Comp_2:   // S393, max time T#10S, warning time T#7S
              R    "KukaRobot3_CtrlDB".sPLCtoROB.User.Cycle.DI307_ScanPartFinish
              N    "KukaRobot3_CtrlDB".sPLCtoROB.User.Cycle.DI306_ScanPartComplete
   END_STEP
   TRANSITION Trans341 FROM RobotScanGripPos2Comp_2 TO WaitRobotScanGripPos3Reach_2   // T392
      := NOT "KukaRobot3_CtrlDB".sROBtoPLC.User.Cycle.DO308_ScanPos2Reach;
   END_TRANSITION
   STEP WaitRobotScanGripPos3Reach_2:   // S394, max time T#10S, warning time T#7S
   END_STEP
   TRANSITION Trans342 FROM WaitRobotScanGripPos3Reach_2 TO "Check reader Ready_21"   // T393
      := "KukaRobot3_CtrlDB".sROBtoPLC.User.Cycle.DO309_ScanPos3Reach;
   END_TRANSITION
   STEP "Check reader Ready_21":   // S395, max time T#10S, warning time T#7S
   END_STEP
   TRANSITION Trans646 FROM "Check reader Ready_21" TO "Start 11st reading_7"   // T649
      := "KeyenceSR1000Ctrl_803A1DB".oReady;
   END_TRANSITION
   STEP "Start 11st reading_7":   // S396, max time T#10S, warning time T#7S
          S1  S    "KeyenceSR1000Ctrl_803A1DB".ioAutoTrigger
   END_STEP
   TRANSITION Trans647 FROM "Start 11st reading_7" TO "Wait reading complete_21"   // T650
      := NOT "KeyenceSR1000Ctrl_803A1DB".sHMI.Status.Ready;
   END_TRANSITION
   STEP "Wait reading complete_21":   // S397, max time T#10S, warning time T#7S
   END_STEP
   TRANSITION ReadOK_22 FROM "Wait reading complete_21" TO DataMove_22   // T394
      := "KeyenceSR1000Ctrl_803A1DB".sHMI.Status.Complete;
   END_TRANSITION
   STEP DataMove_22:   // S398, max time T#10S, warning time T#7S
              N    "AutoProcessData".GripperCode_R3[3]:="KeyenceSR1000Ctrl_803A1DB".sHMI.Status.CurrentCode
   END_STEP
   TRANSITION Trans343 FROM DataMove_22 TO RobotScanGripPos3Comp_2   // T395
      := "AlwaysTRUE";
   END_TRANSITION
   STEP RobotScanGripPos3Comp_2:   // S399, max time T#10S, warning time T#7S
              R    "KukaRobot3_CtrlDB".sPLCtoROB.User.Cycle.DI307_ScanPartFinish
              N    "KukaRobot3_CtrlDB".sPLCtoROB.User.Cycle.DI306_ScanPartComplete
   END_STEP
   TRANSITION Trans344 FROM RobotScanGripPos3Comp_2 TO WaitRobotScanGripPos4Reach_2   // T396
      := NOT "KukaRobot3_CtrlDB".sROBtoPLC.User.Cycle.DO309_ScanPos3Reach;
   END_TRANSITION
   STEP WaitRobotScanGripPos4Reach_2:   // S401, max time T#10S, warning time T#7S
   END_STEP
   TRANSITION Trans345 FROM WaitRobotScanGripPos4Reach_2 TO "Check reader Ready_22"   // T397
      := "KukaRobot3_CtrlDB".sROBtoPLC.User.Cycle.DO310_ScanPos4Reach;
   END_TRANSITION
   STEP "Check reader Ready_22":   // S402, max time T#10S, warning time T#7S
   END_STEP
   TRANSITION Trans648 FROM "Check reader Ready_22" TO "Start 11st reading_8"   // T651
      := "KeyenceSR1000Ctrl_803A1DB".oReady;
   END_TRANSITION
   STEP "Start 11st reading_8":   // S403, max time T#10S, warning time T#7S
          S1  S    "KeyenceSR1000Ctrl_803A1DB".ioAutoTrigger
   END_STEP
   TRANSITION Trans649 FROM "Start 11st reading_8" TO "Wait reading complete_22"   // T652
      := NOT "KeyenceSR1000Ctrl_803A1DB".sHMI.Status.Ready;
   END_TRANSITION
   STEP "Wait reading complete_22":   // S404, max time T#10S, warning time T#7S
   END_STEP
   TRANSITION ReadOK_23 FROM "Wait reading complete_22" TO DataMove_23   // T398
      := "KeyenceSR1000Ctrl_803A1DB".sHMI.Status.Complete;
   END_TRANSITION
   STEP DataMove_23:   // S405, max time T#10S, warning time T#7S
              N    "AutoProcessData".GripperCode_R3[4]:="KeyenceSR1000Ctrl_803A1DB".sHMI.Status.CurrentCode
   END_STEP
   TRANSITION Trans346 FROM DataMove_23 TO RobotScanGripPos4Comp_2   // T399
      := "AlwaysTRUE";
   END_TRANSITION
   STEP RobotScanGripPos4Comp_2:   // S406, max time T#10S, warning time T#7S
              N    "KukaRobot3_CtrlDB".sPLCtoROB.User.Cycle.DI307_ScanPartFinish
              N    "KukaRobot3_CtrlDB".sPLCtoROB.User.Cycle.DI306_ScanPartComplete
   END_STEP
   TRANSITION Trans347 FROM RobotScanGripPos4Comp_2 TO WaitRobot2ScanFinishAndInHome   // T401
      := "KukaRobot3_CtrlDB".sROBtoPLC.User.Cycle.DO306_GripScanFinish;
   END_TRANSITION
   STEP WaitRobot2ScanFinishAndInHome:   // S407, max time T#10S, warning time T#7S
   END_STEP
   TRANSITION Trans371 FROM WaitRobot2ScanFinishAndInHome TO RequestRobotScanFixture   // T402
      := "Robot_DB".Robot_2.GripCompareCodeOK AND "KukaRobot2_CtrlDB".sROBtoPLC.Sys.SO.IN_HOME AND "KukaRobot2_CtrlDB".sROBtoPLC.User.Home.DO181_Robot3Area;
   END_TRANSITION
   STEP Robot3CheckScanStatus:   // S411, max time T#10S, warning time T#7S
   END_STEP
   TRANSITION GripScanNG1 FROM Robot3CheckScanStatus TO RequestRobotScan_1   // T406
      := NOT "AutoProcessData".GlobalData.Robot3GripperCodeOKFlag;
   END_TRANSITION
   TRANSITION GripScanOK FROM Robot3CheckScanStatus TO RequestRobotScanFixture   // T407
      := "AutoProcessData".GlobalData.Robot3GripperCodeOKFlag AND NOT "AutoProcessData".GlobalData.Fixture2CodeOKFlag;
   END_TRANSITION
   TRANSITION ALLScanOk FROM Robot3CheckScanStatus TO Robot3CheckScanResult   // T712
      := "AutoProcessData".GlobalData.Robot3GripperCodeOKFlag AND "AutoProcessData".GlobalData.Fixture2CodeOKFlag;
   END_TRANSITION
   STEP WaitRobotScanPos1Reach_4:   // S412, max time T#10S, warning time T#7S
   END_STEP
   TRANSITION Trans624 FROM WaitRobotScanPos1Reach_4 TO Robot3CheckScanResult   // T653
      := TRUE;
   END_TRANSITION
   STEP "Start 5st reading_2":   // S298, max time T#10S, warning time T#7S
   END_STEP
   TRANSITION Trans349 FROM "Start 5st reading_2" TO "Wait reading complete_23"   // T318
      := TRUE;
   END_TRANSITION
   STEP "Check reader Ready_23":   // S349, max time T#10S, warning time T#7S
   END_STEP
   TRANSITION Trans350 FROM "Check reader Ready_23" TO "Start 5st reading_2"   // T330
      := TRUE;
   END_TRANSITION
   STEP "Wait reading complete_23":   // S413, max time T#10S, warning time T#7S
   END_STEP
   TRANSITION ReadOK_24 FROM "Wait reading complete_23" TO DataMove_24   // T320
      := TRUE;
   END_TRANSITION
   STEP DataMove_24:   // S414, max time T#10S, warning time T#7S
   END_STEP
   TRANSITION Trans348 FROM DataMove_24 TO WaitRobotScanPos1Reach_4   // T328
      := "AlwaysTRUE";
   END_TRANSITION

   // sequencer 6: S700-S710 Robot1_Maintenance Pos
   STEP MaintenanceProcess:   // S700, max time T#10S, warning time T#7S
   END_STEP
   TRANSITION Trans625 FROM MaintenanceProcess TO ReqRobotToMantenPos   // T700
      := "KukaRobot2_CtrlDB".sROBtoPLC.User.Cycle.DO298_MaintainFinish OR "KukaRobot2_CtrlDB".sROBtoPLC.Sys.SO.IN_HOME;
   END_TRANSITION
   STEP ReqRobotToMantenPos:   // S701, max time T#10S, warning time T#7S
              N    "ChangeOver_DB".Robot_1.Req_RobotToMaintenancePos
   END_STEP
   TRANSITION Trans626 FROM ReqRobotToMantenPos TO WaitR1MaintenPosFinsh   // T701
      := "KukaRobot1_CtrlDB".sROBtoPLC.User.Cycle.DO297_MaintainInside;
   END_TRANSITION
   STEP WaitR1MaintenPosFinsh:   // S702, max time T#10S, warning time T#7S
   END_STEP
   TRANSITION Trans627 FROM WaitR1MaintenPosFinsh TO Robot2ToMaintenance   // T702
      := "KukaRobot1_CtrlDB".sROBtoPLC.User.Cycle.DO298_MaintainFinish;
   END_TRANSITION
   STEP Robot2ToMaintenance:   // S704, max time T#10S, warning time T#7S
   END_STEP
   TRANSITION Trans650 FROM Robot2ToMaintenance TO Step720   // T704, jump
      := ("KukaRobot1_CtrlDB".sROBtoPLC.User.Cycle.DO298_MaintainFinish OR "KukaRobot1_CtrlDB".sROBtoPLC.Sys.SO.IN_HOME) AND ("KukaRobot3_CtrlDB".sROBtoPLC.User.Cycle.DO301_HomeFinish OR "KukaRobot3_CtrlDB".sROBtoPLC.Sys.SO.IN_HOME) AND NOT "KukaRobot3_CtrlDB".sROBtoPLC.User.Cycle.DO225_ScanPosInside AND NOT "AutoProcessData".GlobalData.Robot2GripperCodeOKFlag;
   END_TRANSITION

   // sequencer 7: S720-S730 Robot2_Maintenance Pos
   STEP Step720:   // S720, max time T#10S, warning time T#7S
   END_STEP
   TRANSITION Trans720 FROM Step720 TO MaintenanceProcess_1   // T720
      := TRUE;
   END_TRANSITION
   STEP MaintenanceProcess_1:   // S706, max time T#10S, warning time T#7S
   END_STEP
   TRANSITION Trans655 FROM MaintenanceProcess_1 TO ReqRobotToMantenPos_1   // T706
      := ("KukaRobot3_CtrlDB".sROBtoPLC.User.Cycle.DO298_MaintainFinish OR "KukaRobot3_CtrlDB".sROBtoPLC.Sys.SO.IN_HOME) AND NOT "KukaRobot3_CtrlDB".sROBtoPLC.User.Cycle.DO225_ScanPosInside;
   END_TRANSITION
   STEP ReqRobotToMantenPos_1:   // S707, max time T#10S, warning time T#7S
              N    "ChangeOver_DB".Robot_2.Req_RobotToMaintenancePos
   END_STEP
   TRANSITION Trans656 FROM ReqRobotToMantenPos_1 TO WaitR1MaintenPosFinsh_1   // T707
      := "KukaRobot2_CtrlDB".sROBtoPLC.User.Cycle.DO297_MaintainInside;
   END_TRANSITION
   STEP WaitR1MaintenPosFinsh_1:   // S708, max time T#10S, warning time T#7S
   END_STEP
   TRANSITION Trans657 FROM WaitR1MaintenPosFinsh_1 TO Robot3ToMaintenance   // T708
      := "KukaRobot2_CtrlDB".sROBtoPLC.User.Cycle.DO298_MaintainFinish;
   END_TRANSITION
   STEP Robot3ToMaintenance:   // S710, max time T#10S, warning time T#7S
   END_STEP
   TRANSITION Trans659 FROM Robot3ToMaintenance TO Step712   // T710, jump
      := ("KukaRobot2_CtrlDB".sROBtoPLC.User.Cycle.DO298_MaintainFinish OR "KukaRobot2_CtrlDB".sROBtoPLC.Sys.SO.IN_HOME) AND NOT "KukaRobot2_CtrlDB".sROBtoPLC.User.Cycle.DO249_ScanNGPutInside AND NOT "KukaRobot2_CtrlDB".sROBtoPLC.User.Cycle.DO253_GlueNGPutInside AND NOT "KukaRobot2_CtrlDB".sROBtoPLC.User.Cycle.DO273_PressPutPart1Inside AND NOT "AutoProcessData".GlobalData.Robot3GripperCodeOKFlag AND NOT "AutoProcessData".GlobalData.Fixture2CodeOKFlag;
   END_TRANSITION

   // sequencer 8: S740-S750 Robot3_Maintenance Pos
   STEP Step712:   // S740, max time T#10S, warning time T#7S
   END_STEP
   TRANSITION Trans740 FROM Step712 TO MaintenanceProcess_2   // T740
      := TRUE;
   END_TRANSITION
   STEP MaintenanceProcess_2:   // S713, max time T#10S, warning time T#7S
   END_STEP
   TRANSITION Trans661 FROM MaintenanceProcess_2 TO ReqRobotToMantenPos_2   // T713
      := TRUE;
   END_TRANSITION
   STEP ReqRobotToMantenPos_2:   // S714, max time T#10S, warning time T#7S
              N    "ChangeOver_DB".Robot_3.Req_RobotToMaintenancePos
   END_STEP
   TRANSITION Trans662 FROM ReqRobotToMantenPos_2 TO WaitR1MaintenPosFinsh_2   // T714
      := "KukaRobot3_CtrlDB".sROBtoPLC.User.Cycle.DO297_MaintainInside;
   END_TRANSITION
   STEP WaitR1MaintenPosFinsh_2:   // S715, max time T#10S, warning time T#7S
   END_STEP
   TRANSITION Trans663 FROM WaitR1MaintenPosFinsh_2 TO CheckStationEmpty   // T715
      := "KukaRobot3_CtrlDB".sROBtoPLC.User.Cycle.DO298_MaintainFinish;
   END_TRANSITION
   STEP CycleEnd_2:   // S716, max time T#10S, warning time T#7S
              R    "ChangeOver_DB".Global.ChangeOverRequest
   END_STEP
   TRANSITION Trans664 FROM CycleEnd_2 TO END   // T716
      := "AlwaysFALSE";
   END_TRANSITION
   STEP CheckStationEmpty:   // S416, max time T#10S, warning time T#7S
   END_STEP
   TRANSITION Trans413 FROM CheckStationEmpty TO CheckTypeChenge   // T413
      := "ChangeOver_DB".Global.Station_empty AND "AutoProcessControl".Global.ALL_BeltPalletEmptyFinish;
   END_TRANSITION
   STEP CheckTypeChenge:   // S418, max time T#10S, warning time T#7S
   END_STEP
   TRANSITION ChengeOk FROM CheckTypeChenge TO TypeCheckOk   // T415
      := "ST10_RecipeDB".Recipe.Equal AND ("ST10_RecipeDB".Recipe.RecordName <> '');
   END_TRANSITION
   TRANSITION TypeChange FROM CheckTypeChenge TO CheckTypeTrigger   // T417
      := NOT "ST10_RecipeDB".Recipe.Equal AND "ChangeOver_DB".Global.ChangeOverSelected AND "ChangeOver_DB".Global.ChangeOverRequest;
   END_TRANSITION
   STEP TypeCheckOk:   // S419, max time T#10S, warning time T#7S
   END_STEP
   TRANSITION Trans416 FROM TypeCheckOk TO CycleEnd_2   // T416
      := TRUE;
   END_TRANSITION
   STEP CheckTypeTrigger:   // S420, max time T#10S, warning time T#7S
              N    "ChangeOver_DB".Global.ChangeOverActive
   END_STEP
   TRANSITION Trans418 FROM CheckTypeTrigger TO ResetChangeOverReq   // T418
      := "ST10_RecipeDB".Recipe.Equal AND ("ST10_RecipeDB".Recipe.RecordName <> '') AND NOT "ChangeOver_DB".Global.ChangeOverSelected;
   END_TRANSITION
   STEP ResetChangeOverReq:   // S421, max time T#10S, warning time T#7S
              R    "ChangeOver_DB".Global.ChangeOverRequest
   END_STEP
   TRANSITION Trans419 FROM ResetChangeOverReq TO CycleEnd_2   // T419
      := NOT "ChangeOver_DB".Global.ChangeOverSelected AND NOT "ChangeOver_DB".Global.ChangeOverRequest;
   END_TRANSITION

   // permanent post-instructions
   NETWORK 1
      #ioPM_Inface.StepNum := #RT_DATA.S_DISPLAY;
   NETWORK 2
      IF #iSysInface.Reset THEN #AlarmID := 0; END_IF;
   NETWORK 3
      #TON[10].TON(IN := #工件放行中, PT := T#0.5S);
      IF #TON[10].Q THEN #工件放行中 := FALSE; END_IF;
END_FUNCTION_BLOCK
